KUKA KRL program: MyProgram_220().src

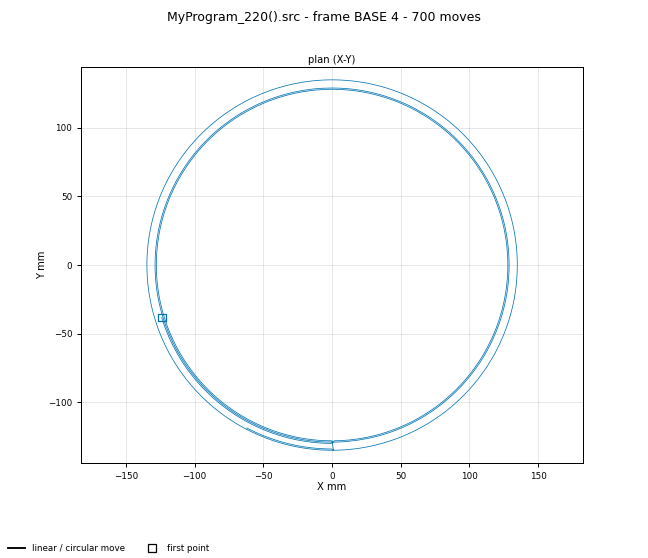
[picture p0: tool path of MyProgram_220().src in frame BASE 4, 700 of 700 moves have a stored position in this frame; points joined in program order, loops and branches not executed]
&ACCESS RVP
&REL 1
&PARAM TEMPLATE = C:\KRC\Roboter\Template\vorgabe
&PARAM EDITMASK = *
DEF MyProgram_220()
; ---- Setting reference (Base) ----
$BASE = BASE_DATA[4]

; --------------------------
; ---- Setting tool (TCP) ----
$TOOL = TOOL_DATA[3]
; --------------------------

$VEL.CP = VEL_APROX_PRINT
Startdeposition()
$VEL.CP = VEL_PRINT
LIN {X -124.0499,Y -38.1824,Z 153,A -164.431,B 20.1252,C -0.668,E1 19.9831,E2 612.3384} C_DIS
LIN {X -122.2235,Y -43.678,Z 153,A -161.8413,B 20.1254,C -0.6617,E1 19.9854,E2 609.7482} C_DIS
LIN {X -120.9472,Y -47.0955,Z 153,A -160.3023,B 20.1256,C -0.6544,E1 19.987,E2 608.2196} C_DIS
LIN {X -119.759,Y -50.0398,Z 153,A -158.8735,B 20.1257,C -0.6515,E1 19.9885,E2 606.7893} C_DIS
LIN {X -118.4765,Y -53.0047,Z 153,A -157.3393,B 20.1257,C -0.6515,E1 19.9902,E2 605.2441} C_DIS
LIN {X -116.9818,Y -56.2275,Z 153,A -155.8456,B 20.1259,C -0.6444,E1 19.992,E2 603.761} C_DIS
LIN {X -115.591,Y -59.0333,Z 153,A -154.3618,B 20.1259,C -0.6444,E1 19.9939,E2 602.2669} C_DIS
LIN {X -112.2722,Y -65.1279,Z 153,A -151.3304,B 20.1262,C -0.635,E1 19.998,E2 599.2428} C_DIS
LIN {X -110.2468,Y -68.5007,Z 153,A -149.5687,B 20.1263,C -0.6315,E1 20.0005,E2 597.48} C_DIS
LIN {X -107.8897,Y -72.1562,Z 153,A -147.8172,B 20.1267,C -0.6202,E1 20.0032,E2 595.7503} C_DIS
LIN {X -106.0602,Y -74.8192,Z 153,A -146.138,B 20.1265,C -0.6263,E1 20.0059,E2 594.0426} C_DIS
LIN {X -103.646,Y -78.1293,Z 153,A -144.4345,B 20.1267,C -0.6179,E1 20.0087,E2 592.3532} C_DIS
LIN {X -101.177,Y -81.3013,Z 153,A -142.5934,B 20.1267,C -0.6163,E1 20.0119,E2 590.5058} C_DIS
LIN {X -99.0599,Y -83.8683,Z 153,A -141.0774,B 20.1268,C -0.6147,E1 20.0146,E2 588.9855} C_DIS
LIN {X -96.3177,Y -87.0039,Z 153,A -139.1751,B 20.1268,C -0.6131,E1 20.0182,E2 587.0772} C_DIS
LIN {X -93.3696,Y -90.16,Z 153,A -137.2715,B 20.127,C -0.6089,E1 20.0218,E2 585.1754} C_DIS
LIN {X -88.6302,Y -94.8219,Z 153,A -134.3468,B 20.1272,C -0.6024,E1 20.0277,E2 582.254} C_DIS
LIN {X -86.2647,Y -96.9806,Z 153,A -132.8941,B 20.1272,C -0.6012,E1 20.0307,E2 580.7976} C_DIS
LIN {X -82.9316,Y -99.8452,Z 153,A -130.925,B 20.1272,C -0.5986,E1 20.0349,E2 578.8263} C_DIS
LIN {X -79.669,Y -102.4674,Z 153,A -129.0942,B 20.1274,C -0.5947,E1 20.0389,E2 576.9986} C_DIS
LIN {X -76.0312,Y -105.1949,Z 153,A -126.47,B 20.1268,C -0.6155,E1 20.045,E2 574.3017} C_DIS
LIN {X -71.6372,Y -108.2354,Z 153,A -125.0313,B 20.1279,C -0.5755,E1 20.0481,E2 572.9738} C_DIS
LIN {X -65.749,Y -111.9096,Z 153,A -121.6773,B 20.1278,C -0.5823,E1 20.0562,E2 569.5867} C_DIS
LIN {X -61.9654,Y -114.0484,Z 153,A -119.6951,B 20.1278,C -0.5822,E1 20.061,E2 567.5976} C_DIS
LIN {X -58.1719,Y -116.0295,Z 153,A -117.7274,B 20.1278,C -0.5829,E1 20.0659,E2 565.621} C_DIS
LIN {X -53.9421,Y -118.0541,Z 153,A -115.5017,B 20.1276,C -0.5867,E1 20.0716,E2 563.377} C_DIS
LIN {X -50.8123,Y -119.4344,Z 153,A -113.9211,B 20.1276,C -0.588,E1 20.0757,E2 561.7882} C_DIS
LIN {X -47.3478,Y -120.8491,Z 153,A -112.8761,B 20.1283,C -0.5621,E1 20.0782,E2 560.8158} C_DIS
LIN {X -43.644,Y -122.2357,Z 153,A -110.9408,B 20.1281,C -0.568,E1 20.0834,E2 558.8581} C_DIS
LIN {X -40.3205,Y -123.3734,Z 153,A -109.2108,B 20.128,C -0.574,E1 20.088,E2 557.1068} C_DIS
LIN {X -36.084,Y -124.6769,Z 153,A -107.4194,B 20.1282,C -0.5659,E1 20.0927,E2 555.335} C_DIS
LIN {X -32.6503,Y -125.6214,Z 153,A -105.6991,B 20.1281,C -0.5709,E1 20.0974,E2 553.5969} C_DIS
LIN {X -28.2074,Y -126.6929,Z 153,A -103.5651,B 20.128,C -0.5746,E1 20.1033,E2 551.4486} C_DIS
LIN {X -23.1298,Y -127.7159,Z 153,A -100.8212,B 20.1275,C -0.5924,E1 20.111,E2 548.6491} C_DIS
LIN {X -17.8854,Y -128.5559,Z 153,A -98.8039,B 20.1279,C -0.5784,E1 20.1164,E2 546.6708} C_DIS
LIN {X -14.3127,Y -129.0024,Z 153,A -97.7565,B 20.1285,C -0.5559,E1 20.1192,E2 545.6878} C_DIS
LIN {X -9.5222,Y -129.4436,Z 153,A -95.2617,B 20.1281,C -0.5709,E1 20.1262,E2 543.1478} C_DIS
LIN {X -4.67,Y -129.7099,Z 153,A -93.267,B 20.1282,C -0.5648,E1 20.1317,E2 541.1703} C_DIS
LIN {X -0.7047,Y -129.7915,Z 153,A -91.6167,B 20.1283,C -0.561,E1 20.1363,E2 539.5311} C_DIS
LIN {X -0.7047,Y -129.7915,Z 153,A -91.6167,B 20.1283,C -0.561,E1 20.1363,E2 539.5311} C_DIS
Enddeposition()
LIN {X 0.8922,Y -128.8473,Z 153,A -90.561,B 18.6911,C -0.3834,E1 18.6972,E2 538.8726} C_DIS
Startdeposition()
$VEL.CP = VEL_PRINT
LIN {X -1.7978,Y -128.8411,Z 153,A -92.3931,B 18.6916,C -0.3592,E1 18.6919,E2 540.7802} C_DIS
LIN {X -4.9626,Y -128.7576,Z 153,A -94.0816,B 18.6918,C -0.3487,E1 18.6871,E2 542.502} C_DIS
LIN {X -8.6262,Y -128.566,Z 153,A -95.4711,B 18.6916,C -0.3576,E1 18.6833,E2 543.8641} C_DIS
LIN {X -11.8778,Y -128.3052,Z 153,A -97.4568,B 18.692,C -0.3381,E1 18.6776,E2 545.9123} C_DIS
LIN {X -16.8123,Y -127.7516,Z 153,A -99.0184,B 18.6915,C -0.3623,E1 18.6735,E2 547.3997} C_DIS
LIN {X -20.6153,Y -127.1946,Z 153,A -100.8214,B 18.6915,C -0.3593,E1 18.6684,E2 549.2142} C_DIS
LIN {X -23.6637,Y -126.6626,Z 153,A -102.3077,B 18.6916,C -0.3558,E1 18.6643,E2 550.7136} C_DIS
LIN {X -28.0145,Y -125.7726,Z 153,A -104.178,B 18.6916,C -0.3606,E1 18.6593,E2 552.5722} C_DIS
LIN {X -31.1189,Y -125.0401,Z 153,A -105.392,B 18.6914,C -0.3688,E1 18.656,E2 553.7625} C_DIS
LIN {X -34.3257,Y -124.1972,Z 153,A -106.9978,B 18.6914,C -0.365,E1 18.6516,E2 555.3838} C_DIS
LIN {X -37.1865,Y -123.3714,Z 153,A -108.3483,B 18.6914,C -0.365,E1 18.648,E2 556.7375} C_DIS
LIN {X -40.6641,Y -122.2681,Z 153,A -109.8927,B 18.6914,C -0.3691,E1 18.6439,E2 558.2728} C_DIS
LIN {X -43.8363,Y -121.167,Z 153,A -111.4208,B 18.6914,C -0.3691,E1 18.6399,E2 559.8049} C_DIS
LIN {X -50.8161,Y -118.4097,Z 153,A -114.8178,B 18.6914,C -0.3702,E1 18.6311,E2 563.2088} C_DIS
LIN {X -54.652,Y -116.69,Z 153,A -116.9427,B 18.6915,C -0.3631,E1 18.6256,E2 565.363} C_DIS
LIN {X -59.4438,Y -114.3228,Z 153,A -119.0566,B 18.6913,C -0.3755,E1 18.6204,E2 567.4459} C_DIS
LIN {X -63.0684,Y -112.365,Z 153,A -120.8296,B 18.6912,C -0.38,E1 18.6161,E2 569.2117} C_DIS
LIN {X -67.2669,Y -109.9031,Z 153,A -123.1372,B 18.6912,C -0.378,E1 18.6105,E2 571.5353} C_DIS
LIN {X -71.1021,Y -107.462,Z 153,A -125.0591,B 18.6911,C -0.3847,E1 18.6061,E2 573.445} C_DIS
LIN {X -74.9299,Y -104.8285,Z 153,A -127.1982,B 18.6911,C -0.3854,E1 18.6012,E2 575.5916} C_DIS
LIN {X -78.3456,Y -102.3009,Z 153,A -128.9712,B 18.6909,C -0.3928,E1 18.5972,E2 577.3502} C_DIS
LIN {X -81.75,Y -99.6018,Z 153,A -131.0814,B 18.6909,C -0.39,E1 18.5926,E2 579.4801} C_DIS
LIN {X -85.1235,Y -96.7346,Z 153,A -132.9003,B 18.6909,C -0.399,E1 18.5888,E2 581.2806} C_DIS
LIN {X -91.5255,Y -90.7005,Z 153,A -136.9673,B 18.6908,C -0.4014,E1 18.5806,E2 585.3631} C_DIS
LIN {X -94.7022,Y -87.3787,Z 153,A -139.0611,B 18.6908,C -0.4041,E1 18.5765,E2 587.4613} C_DIS
LIN {X -97.6736,Y -84.0439,Z 153,A -141.0409,B 18.6906,C -0.4087,E1 18.5729,E2 589.4388} C_DIS
LIN {X -101.5319,Y -79.3402,Z 153,A -143.629,B 18.6904,C -0.419,E1 18.5684,E2 592.0113} C_DIS
LIN {X -103.7936,Y -76.357,Z 153,A -145.4466,B 18.6904,C -0.4177,E1 18.5653,E2 593.845} C_DIS
LIN {X -106.3954,Y -72.6884,Z 153,A -147.4209,B 18.6903,C -0.4234,E1 18.5621,E2 595.8146} C_DIS
LIN {X -108.6997,Y -69.1953,Z 153,A -149.3063,B 18.6903,C -0.4273,E1 18.5593,E2 597.7011} C_DIS
LIN {X -110.9258,Y -65.5675,Z 153,A -151.256,B 18.6901,C -0.4302,E1 18.5565,E2 599.6554} C_DIS
LIN {X -112.4474,Y -62.9218,Z 153,A -152.7042,B 18.6901,C -0.4306,E1 18.5545,E2 601.1128} C_DIS
LIN {X -114.4576,Y -59.1871,Z 153,A -154.5413,B 18.69,C -0.4373,E1 18.5521,E2 602.9423} C_DIS
LIN {X -116.1156,Y -55.8596,Z 153,A -155.9219,B 18.6897,C -0.4511,E1 18.5504,E2 604.2898} C_DIS
LIN {X -117.4691,Y -52.9543,Z 153,A -157.4356,B 18.6897,C -0.452,E1 18.5486,E2 605.8121} C_DIS
LIN {X -118.5866,Y -50.407,Z 153,A -158.9047,B 18.6897,C -0.4475,E1 18.547,E2 607.3065} C_DIS
LIN {X -119.9416,Y -47.0875,Z 153,A -160.199,B 18.6894,C -0.4622,E1 18.5457,E2 608.5646} C_DIS
LIN {X -121.0477,Y -44.1669,Z 153,A -161.8114,B 18.6894,C -0.4586,E1 18.5441,E2 610.2009} C_DIS
LIN {X -122.7867,Y -39.0704,Z 153,A -164.1851,B 18.6894,C -0.4662,E1 18.542,E2 612.5694} C_DIS
LIN {X -123.9311,Y -35.2775,Z 153,A -165.9601,B 18.6892,C -0.4709,E1 18.5406,E2 614.3438} C_DIS
LIN {X -124.8345,Y -31.9292,Z 153,A -167.5525,B 18.6892,C -0.4738,E1 18.5395,E2 615.9399} C_DIS
LIN {X -125.8011,Y -27.8864,Z 153,A -169.46,B 18.689,C -0.4773,E1 18.5383,E2 617.8519} C_DIS
LIN {X -126.5739,Y -24.1273,Z 153,A -171.1769,B 18.689,C -0.4821,E1 18.5373,E2 619.5676} C_DIS
LIN {X -127.2655,Y -20.1692,Z 153,A -172.7668,B 18.6886,C -0.4941,E1 18.5366,E2 621.1327} C_DIS
LIN {X -127.7311,Y -16.968,Z 153,A -174.4022,B 18.6886,C -0.4919,E1 18.536,E2 622.7886} C_DIS
LIN {X -128.1554,Y -13.3956,Z 153,A -176.0902,B 18.6886,C -0.4938,E1 18.5354,E2 624.4845} C_DIS
LIN {X -128.5161,Y -9.3142,Z 153,A -177.7957,B 18.6884,C -0.5034,E1 18.5351,E2 626.1742} C_DIS
LIN {X -128.7367,Y -5.4997,Z 153,A -179.3666,B 18.6881,C -0.5129,E1 18.5348,E2 627.7281} C_DIS
LIN {X -128.8292,Y -2.5182,Z 153,A 179.1207,B 18.6881,C -0.5108,E1 18.5348,E2 629.2602} C_DIS
LIN {X -128.8489,Y 1.1038,Z 153,A 177.6722,B 18.6879,C -0.5212,E1 18.5348,E2 630.6879} C_DIS
LIN {X -128.792,Y 3.9938,Z 153,A 176.1149,B 18.688,C -0.5161,E1 18.5348,E2 632.2743} C_DIS
LIN {X -128.5815,Y 8.3752,Z 153,A 173.9578,B 18.688,C -0.5152,E1 18.5352,E2 634.4519} C_DIS
LIN {X -128.3292,Y 11.6281,Z 153,A 172.6535,B 18.6878,C -0.5246,E1 18.5355,E2 635.7376} C_DIS
LIN {X -127.8595,Y 15.9868,Z 153,A 170.6979,B 18.6877,C -0.5304,E1 18.5361,E2 637.691} C_DIS
LIN {X -127.3978,Y 19.3149,Z 153,A 169.2335,B 18.6875,C -0.536,E1 18.5367,E2 639.1497} C_DIS
LIN {X -126.6839,Y 23.5521,Z 153,A 167.3093,B 18.6874,C -0.5415,E1 18.5377,E2 641.0727} C_DIS
LIN {X -125.9625,Y 27.1388,Z 153,A 165.7576,B 18.6871,C -0.549,E1 18.5385,E2 642.6134} C_DIS
LIN {X -125.0826,Y 30.9515,Z 153,A 163.8735,B 18.6871,C -0.5494,E1 18.5398,E2 644.5113} C_DIS
LIN {X -123.9507,Y 35.2073,Z 153,A 161.3522,B 18.6875,C -0.5367,E1 18.5417,E2 647.0929} C_DIS
LIN {X -122.4844,Y 40.0115,Z 153,A 159.7319,B 18.6867,C -0.5638,E1 18.543,E2 648.6408} C_DIS
LIN {X -121.2971,Y 43.4752,Z 153,A 158.0558,B 18.6867,C -0.567,E1 18.5446,E2 650.3199} C_DIS
LIN {X -119.855,Y 47.3102,Z 153,A 156.2801,B 18.6864,C -0.5739,E1 18.5464,E2 652.0876} C_DIS
LIN {X -118.5641,Y 50.4591,Z 153,A 154.6433,B 18.6864,C -0.5742,E1 18.5481,E2 653.7362} C_DIS
LIN {X -117.0382,Y 53.8991,Z 153,A 152.5033,B 18.6867,C -0.5634,E1 18.5507,E2 655.9261} C_DIS
LIN {X -115.0458,Y 58.0318,Z 153,A 151.1702,B 18.6858,C -0.5929,E1 18.5522,E2 657.1765} C_DIS
LIN {X -113.5082,Y 60.9869,Z 153,A 149.4584,B 18.686,C -0.5893,E1 18.5545,E2 658.9123} C_DIS
LIN {X -111.3388,Y 64.8638,Z 153,A 147.5706,B 18.6857,C -0.5977,E1 18.5571,E2 660.7873} C_DIS
LIN {X -107.9641,Y 70.337,Z 153,A 144.6774,B 18.6855,C -0.6042,E1 18.5614,E2 663.6801} C_DIS
LIN {X -105.8908,Y 73.4213,Z 153,A 142.8887,B 18.6855,C -0.604,E1 18.5642,E2 665.4818} C_DIS
LIN {X -103.5804,Y 76.647,Z 153,A 141.0878,B 18.6854,C -0.6073,E1 18.5672,E2 667.2843} C_DIS
LIN {X -100.8812,Y 80.1655,Z 153,A 139.1659,B 18.6852,C -0.614,E1 18.5704,E2 669.1977} C_DIS
LIN {X -98.2339,Y 83.3883,Z 153,A 137.2838,B 18.6851,C -0.6177,E1 18.5738,E2 671.0803} C_DIS
LIN {X -95.3863,Y 86.6312,Z 153,A 135.3556,B 18.6849,C -0.622,E1 18.5774,E2 673.0069} C_DIS
LIN {X -92.3221,Y 89.8903,Z 153,A 133.3182,B 18.6849,C -0.625,E1 18.5813,E2 675.047} C_DIS
LIN {X -89.3268,Y 92.8677,Z 153,A 131.4363,B 18.6847,C -0.6291,E1 18.5851,E2 676.9269} C_DIS
LIN {X -86.4368,Y 95.5627,Z 153,A 129.7432,B 18.6845,C -0.6352,E1 18.5885,E2 678.6103} C_DIS
LIN {X -83.4105,Y 98.2151,Z 153,A 127.9104,B 18.6845,C -0.6375,E1 18.5924,E2 680.4457} C_DIS
LIN {X -80.1785,Y 100.8708,Z 153,A 126.018,B 18.6843,C -0.6402,E1 18.5965,E2 682.3394} C_DIS
LIN {X -76.6483,Y 103.5794,Z 153,A 123.9948,B 18.6843,C -0.6426,E1 18.6011,E2 684.3652} C_DIS
LIN {X -74.3543,Y 105.2376,Z 153,A 122.5318,B 18.6844,C -0.6379,E1 18.6044,E2 685.8496} C_DIS
LIN {X -71.6808,Y 107.0766,Z 153,A 120.9403,B 18.6844,C -0.6355,E1 18.6082,E2 687.4562} C_DIS
LIN {X -68.3675,Y 109.222,Z 153,A 119.4648,B 18.6841,C -0.6482,E1 18.6116,E2 688.8982} C_DIS
LIN {X -64.3417,Y 111.641,Z 153,A 117.4252,B 18.6839,C -0.6534,E1 18.6165,E2 690.9298} C_DIS
LIN {X -60.6816,Y 113.6722,Z 153,A 115.6579,B 18.6837,C -0.6597,E1 18.6208,E2 692.6845} C_DIS
LIN {X -57.2859,Y 115.4185,Z 153,A 113.919,B 18.6837,C -0.6609,E1 18.6251,E2 694.426} C_DIS
LIN {X -53.7581,Y 117.1034,Z 153,A 112.164,B 18.6836,C -0.6628,E1 18.6295,E2 696.1811} C_DIS
LIN {X -50.4862,Y 118.5524,Z 153,A 110.6594,B 18.6834,C -0.668,E1 18.6334,E2 697.6743} C_DIS
LIN {X -47.2881,Y 119.8636,Z 153,A 108.9988,B 18.6834,C -0.6656,E1 18.6377,E2 699.3474} C_DIS
LIN {X -43.8521,Y 121.1613,Z 153,A 107.4552,B 18.6834,C -0.6707,E1 18.6417,E2 700.8793} C_DIS
LIN {X -40.8666,Y 122.2006,Z 153,A 106.1838,B 18.6831,C -0.6771,E1 18.645,E2 702.1342} C_DIS
LIN {X -38.5993,Y 122.9372,Z 153,A 104.8373,B 18.6834,C -0.668,E1 18.6487,E2 703.5122} C_DIS
LIN {X -35.0688,Y 123.9894,Z 153,A 103.459,B 18.683,C -0.6789,E1 18.6523,E2 704.8597} C_DIS
LIN {X -32.3809,Y 124.7198,Z 153,A 101.839,B 18.6835,C -0.6664,E1 18.6568,E2 706.5219} C_DIS
LIN {X -27.7778,Y 125.8246,Z 153,A 99.5881,B 18.6835,C -0.663,E1 18.663,E2 708.7876} C_DIS
LIN {X -24.3768,Y 126.5262,Z 153,A 98.4114,B 18.6831,C -0.6772,E1 18.6661,E2 709.9215} C_DIS
LIN {X -20.9195,Y 127.1438,Z 153,A 96.8722,B 18.6831,C -0.6791,E1 18.6703,E2 711.4571} C_DIS
LIN {X -14.7385,Y 128.0085,Z 153,A 94.1208,B 18.6829,C -0.6814,E1 18.6779,E2 714.204} C_DIS
LIN {X -11.298,Y 128.3575,Z 153,A 92.0352,B 18.6836,C -0.6623,E1 18.6839,E2 716.3507} C_DIS
LIN {X -7.0803,Y 128.6599,Z 153,A 90.7429,B 18.6828,C -0.6841,E1 18.6873,E2 717.5754} C_DIS
LIN {X 0.1516,Y 128.8544,Z 153,A 86.6454,B 18.6839,C -0.6528,E1 18.699,E2 721.7707} C_DIS
LIN {X 5.794,Y 128.7246,Z 153,A 84.9882,B 18.6829,C -0.6838,E1 18.7034,E2 723.3306} C_DIS
LIN {X 11.8096,Y 128.3118,Z 153,A 82.0309,B 18.6832,C -0.6734,E1 18.7117,E2 726.3183} C_DIS
LIN {X 16.2936,Y 127.8195,Z 153,A 80.2191,B 18.683,C -0.6801,E1 18.7166,E2 728.1075} C_DIS
LIN {X 19.5858,Y 127.3559,Z 153,A 78.8596,B 18.6828,C -0.684,E1 18.7203,E2 729.4529} C_DIS
LIN {X 23.1661,Y 126.7543,Z 153,A 77.167,B 18.683,C -0.6805,E1 18.725,E2 731.1541} C_DIS
LIN {X 27.1118,Y 125.9684,Z 153,A 75.6191,B 18.6827,C -0.6886,E1 18.7292,E2 732.6741} C_DIS
LIN {X 30.0875,Y 125.2909,Z 153,A 73.9169,B 18.6832,C -0.6749,E1 18.7339,E2 734.4156} C_DIS
LIN {X 33.9159,Y 124.3114,Z 153,A 72.277,B 18.6831,C -0.6781,E1 18.7383,E2 736.0419} C_DIS
LIN {X 36.8949,Y 123.4598,Z 153,A 70.7652,B 18.6833,C -0.6721,E1 18.7424,E2 737.569} C_DIS
LIN {X 40.5844,Y 122.2946,Z 153,A 69.2515,B 18.683,C -0.6784,E1 18.7464,E2 739.0589} C_DIS
LIN {X 43.0947,Y 121.4343,Z 153,A 66.983,B 18.6845,C -0.6366,E1 18.7527,E2 741.4511} C_DIS
LIN {X 49.3151,Y 119.0427,Z 153,A 65.0437,B 18.6833,C -0.6719,E1 18.7574,E2 743.2745} C_DIS
LIN {X 53.1423,Y 117.385,Z 153,A 63.1989,B 18.6833,C -0.6702,E1 18.7621,E2 745.1185} C_DIS
LIN {X 56.4826,Y 115.8148,Z 153,A 61.4722,B 18.6835,C -0.6649,E1 18.7665,E2 746.8553} C_DIS
LIN {X 60.0312,Y 114.0144,Z 153,A 59.931,B 18.6833,C -0.6713,E1 18.7702,E2 748.3707} C_DIS
LIN {X 66.8158,Y 110.178,Z 153,A 56.2335,B 18.6838,C -0.6575,E1 18.7793,E2 752.096} C_DIS
LIN {X 71.3155,Y 107.3204,Z 153,A 53.8497,B 18.6839,C -0.6532,E1 18.7848,E2 754.4823} C_DIS
LIN {X 74.8349,Y 104.8964,Z 153,A 51.9744,B 18.6839,C -0.651,E1 18.7891,E2 756.3555} C_DIS
LIN {X 78.4833,Y 102.1956,Z 153,A 49.9711,B 18.6841,C -0.6481,E1 18.7936,E2 758.358} C_DIS
LIN {X 81.766,Y 99.5887,Z 153,A 48.15,B 18.6841,C -0.6463,E1 18.7975,E2 760.1752} C_DIS
LIN {X 85.0534,Y 96.7966,Z 153,A 46.2322,B 18.6843,C -0.6426,E1 18.8016,E2 762.094} C_DIS
LIN {X 88.3958,Y 93.7533,Z 153,A 44.1218,B 18.6845,C -0.6347,E1 18.8059,E2 764.2172} C_DIS
LIN {X 91.755,Y 90.469,Z 153,A 42.1091,B 18.6845,C -0.6333,E1 18.8099,E2 766.2225} C_DIS
LIN {X 94.6799,Y 87.403,Z 153,A 40.2376,B 18.6847,C -0.6297,E1 18.8135,E2 768.0939} C_DIS
LIN {X 97.4633,Y 84.2881,Z 153,A 38.3922,B 18.6848,C -0.626,E1 18.8169,E2 769.9393} C_DIS
LIN {X 100.483,Y 80.6645,Z 153,A 36.3264,B 18.6849,C -0.6224,E1 18.8205,E2 772.0032} C_DIS
LIN {X 103.11,Y 77.2786,Z 153,A 34.5596,B 18.6849,C -0.6233,E1 18.8235,E2 773.7555} C_DIS
LIN {X 107.3136,Y 71.3258,Z 153,A 31.2168,B 18.6853,C -0.6112,E1 18.8289,E2 777.1132} C_DIS
LIN {X 109.1635,Y 68.4615,Z 153,A 29.4966,B 18.6856,C -0.5993,E1 18.8315,E2 778.8584} C_DIS
LIN {X 110.8629,Y 65.6738,Z 153,A 28.3684,B 18.6854,C -0.6083,E1 18.833,E2 779.9506} C_DIS
LIN {X 112.8659,Y 62.1682,Z 153,A 26.4796,B 18.6856,C -0.5999,E1 18.8356,E2 781.8521} C_DIS
LIN {X 114.5817,Y 58.9434,Z 153,A 25.0921,B 18.6855,C -0.605,E1 18.8374,E2 783.2138} C_DIS
LIN {X 117.1547,Y 53.6472,Z 153,A 22.2619,B 18.686,C -0.5893,E1 18.8409,E2 786.0715} C_DIS
LIN {X 118.447,Y 50.7298,Z 153,A 20.6234,B 18.6863,C -0.5766,E1 18.8427,E2 787.737} C_DIS
LIN {X 119.7997,Y 47.4516,Z 153,A 19.3063,B 18.6862,C -0.5825,E1 18.844,E2 789.026} C_DIS
LIN {X 120.9848,Y 44.3414,Z 153,A 17.7597,B 18.6864,C -0.5756,E1 18.8455,E2 790.582} C_DIS
LIN {X 122.342,Y 40.4419,Z 153,A 16.1053,B 18.6864,C -0.5776,E1 18.847,E2 792.2176} C_DIS
LIN {X 123.5409,Y 36.6179,Z 153,A 14.3858,B 18.6864,C -0.5748,E1 18.8484,E2 793.9319} C_DIS
LIN {X 124.3314,Y 33.8407,Z 153,A 12.9628,B 18.6867,C -0.5655,E1 18.8495,E2 795.3728} C_DIS
LIN {X 125.261,Y 30.2117,Z 153,A 10.9903,B 18.6872,C -0.5482,E1 18.8508,E2 797.383} C_DIS
LIN {X 126.135,Y 26.3337,Z 153,A 9.6959,B 18.6868,C -0.5619,E1 18.8515,E2 798.6248} C_DIS
LIN {X 126.7331,Y 23.2846,Z 153,A 8.2849,B 18.6869,C -0.5565,E1 18.8523,E2 800.041} C_DIS
LIN {X 127.2322,Y 20.3842,Z 153,A 6.5211,B 18.6876,C -0.5343,E1 18.8531,E2 801.8594} C_DIS
LIN {X 127.8062,Y 16.3951,Z 153,A 5.2549,B 18.6871,C -0.5499,E1 18.8535,E2 803.0669} C_DIS
LIN {X 128.5105,Y 9.3908,Z 153,A 2.4485,B 18.6871,C -0.5533,E1 18.8543,E2 805.8399} C_DIS
LIN {X 128.8357,Y 2.1236,Z 153,A -0.7464,B 18.6873,C -0.5448,E1 18.8547,E2 809.035} C_DIS
LIN {X 128.7821,Y -4.335,Z 153,A -4.0261,B 18.688,C -0.5193,E1 18.8546,E2 812.3668} C_DIS
LIN {X 128.3422,Y -11.4815,Z 153,A -7.2602,B 18.6883,C -0.5074,E1 18.8539,E2 815.6115} C_DIS
LIN {X 127.8619,Y -15.9669,Z 153,A -9.1185,B 18.6883,C -0.5071,E1 18.8533,E2 817.4555} C_DIS
LIN {X 127.4527,Y -18.9583,Z 153,A -10.6936,B 18.6886,C -0.4935,E1 18.8527,E2 819.0598} C_DIS
LIN {X 126.6103,Y -23.9373,Z 153,A -12.5459,B 18.6884,C -0.5025,E1 18.8518,E2 820.8695} C_DIS
LIN {X 125.8028,Y -27.8786,Z 153,A -14.5783,B 18.6888,C -0.4871,E1 18.8506,E2 822.9332} C_DIS
LIN {X 125.0008,Y -31.2738,Z 153,A -15.8685,B 18.6886,C -0.493,E1 18.8498,E2 824.1952} C_DIS
LIN {X 124.0369,Y -34.899,Z 153,A -17.399,B 18.6886,C -0.4934,E1 18.8487,E2 825.712} C_DIS
LIN {X 122.9845,Y -38.4507,Z 153,A -19.4112,B 18.6891,C -0.4737,E1 18.847,E2 827.7696} C_DIS
LIN {X 121.5142,Y -42.8698,Z 153,A -21.2595,B 18.6891,C -0.4765,E1 18.8454,E2 829.595} C_DIS
LIN {X 119.7651,Y -47.5376,Z 153,A -23.4411,B 18.6891,C -0.4713,E1 18.8432,E2 831.7759} C_DIS
LIN {X 118.3665,Y -50.916,Z 153,A -24.8633,B 18.6891,C -0.4748,E1 18.8417,E2 833.1766} C_DIS
LIN {X 117.1454,Y -53.6672,Z 153,A -26.5105,B 18.6895,C -0.4584,E1 18.8398,E2 834.8622} C_DIS
LIN {X 115.2522,Y -57.623,Z 153,A -28.7299,B 18.6899,C -0.442,E1 18.837,E2 837.116} C_DIS
LIN {X 113.6154,Y -60.7873,Z 153,A -30.032,B 18.6897,C -0.4488,E1 18.8353,E2 838.3875} C_DIS
LIN {X 111.463,Y -64.6492,Z 153,A -31.9535,B 18.6898,C -0.4451,E1 18.8327,E2 840.3067} C_DIS
LIN {X 109.2277,Y -68.3587,Z 153,A -33.9322,B 18.69,C -0.4377,E1 18.8298,E2 842.2945} C_DIS
LIN {X 106.9157,Y -71.9213,Z 153,A -35.806,B 18.69,C -0.4332,E1 18.8269,E2 844.1694} C_DIS
LIN {X 104.784,Y -74.9922,Z 153,A -37.4446,B 18.6901,C -0.4298,E1 18.8242,E2 845.8077} C_DIS
LIN {X 102.5622,Y -78.004,Z 153,A -39.1097,B 18.6902,C -0.4255,E1 18.8214,E2 847.4753} C_DIS
LIN {X 99.6794,Y -81.655,Z 153,A -41.0674,B 18.6902,C -0.4246,E1 18.818,E2 849.423} C_DIS
LIN {X 97.3996,Y -84.3615,Z 153,A -42.7538,B 18.6904,C -0.4162,E1 18.8149,E2 851.1248} C_DIS
LIN {X 94.1796,Y -87.9416,Z 153,A -44.7963,B 18.6904,C -0.415,E1 18.8111,E2 853.1587} C_DIS
LIN {X 91.1521,Y -91.0765,Z 153,A -46.6426,B 18.6904,C -0.4141,E1 18.8075,E2 854.997} C_DIS
LIN {X 88.6923,Y -93.4731,Z 153,A -48.2764,B 18.6907,C -0.4064,E1 18.8042,E2 856.6454} C_DIS
LIN {X 85.4273,Y -96.466,Z 153,A -50.1588,B 18.6907,C -0.4055,E1 18.8003,E2 858.5202} C_DIS
LIN {X 82.6432,Y -98.8618,Z 153,A -51.8268,B 18.6907,C -0.4006,E1 18.7967,E2 860.1944} C_DIS
LIN {X 79.8799,Y -101.108,Z 153,A -53.5052,B 18.6909,C -0.3936,E1 18.7931,E2 861.886} C_DIS
LIN {X 75.9801,Y -104.0705,Z 153,A -55.5271,B 18.6909,C -0.3953,E1 18.7886,E2 863.8924} C_DIS
LIN {X 72.5224,Y -106.5088,Z 153,A -57.4849,B 18.691,C -0.3887,E1 18.784,E2 865.8615} C_DIS
LIN {X 68.6992,Y -109.0135,Z 153,A -59.4393,B 18.691,C -0.3881,E1 18.7795,E2 867.8091} C_DIS
LIN {X 65.0563,Y -111.2261,Z 153,A -61.3563,B 18.6911,C -0.3839,E1 18.7749,E2 869.7309} C_DIS
LIN {X 61.4641,Y -113.2508,Z 153,A -63.5586,B 18.6914,C -0.3665,E1 18.7694,E2 871.9784} C_DIS
LIN {X 57.8986,Y -115.1136,Z 153,A -64.8895,B 18.6912,C -0.3815,E1 18.7662,E2 873.2577} C_DIS
LIN {X 54.8571,Y -116.5945,Z 153,A -66.4013,B 18.6912,C -0.3789,E1 18.7624,E2 874.7721} C_DIS
LIN {X 51.9098,Y -117.9363,Z 153,A -67.768,B 18.6912,C -0.3797,E1 18.7589,E2 876.1316} C_DIS
LIN {X 47.9256,Y -119.6087,Z 153,A -69.813,B 18.6913,C -0.3723,E1 18.7536,E2 878.1931} C_DIS
LIN {X 44.2185,Y -121.0291,Z 153,A -71.4368,B 18.6913,C -0.3756,E1 18.7494,E2 879.802} C_DIS
LIN {X 41.1968,Y -122.0906,Z 153,A -73.339,B 18.6917,C -0.3555,E1 18.7442,E2 881.7614} C_DIS
LIN {X 37.4971,Y -123.2764,Z 153,A -74.5826,B 18.6913,C -0.3722,E1 18.741,E2 882.95} C_DIS
LIN {X 34.0113,Y -124.2852,Z 153,A -76.3773,B 18.6915,C -0.3636,E1 18.7361,E2 884.7674} C_DIS
LIN {X 30.2742,Y -125.246,Z 153,A -78.3876,B 18.6917,C -0.3508,E1 18.7306,E2 886.8134} C_DIS
LIN {X 26.309,Y -126.14,Z 153,A -79.8338,B 18.6915,C -0.363,E1 18.7267,E2 888.219} C_DIS
LIN {X 17.449,Y -127.6681,Z 153,A -83.6764,B 18.6915,C -0.3661,E1 18.7162,E2 892.0464} C_DIS
LIN {X 9.4408,Y -128.5068,Z 153,A -87.3874,B 18.6915,C -0.3594,E1 18.7059,E2 895.775} C_DIS
LIN {X 4.7553,Y -128.7657,Z 153,A -89.4989,B 18.6916,C -0.3578,E1 18.6999,E2 897.8906} C_DIS
LIN {X 0.8922,Y -128.8473,Z 153,A -90.5575,B 18.6911,C -0.3823,E1 18.6972,E2 898.8726} C_DIS
Enddeposition()
LIN {X 0.8922,Y -128.8473,Z 153,A -90.5575,B 18.6911,C -0.3823,E1 18.6972,E2 898.8726} C_DIS
Startdeposition()
$VEL.CP = VEL_PRINT
LIN {X 1.5624,Y -127.9047,Z 153,A -89.64,B 17.5227,C -0.2683,E1 17.5287,E2 898.2231} C_DIS
LIN {X 6.2751,Y -127.7591,Z 153,A -87.8027,B 17.5227,C -0.2592,E1 17.5337,E2 896.4169} C_DIS
LIN {X 9.4059,Y -127.5667,Z 153,A -86.3309,B 17.5227,C -0.2621,E1 17.5379,E2 894.9364} C_DIS
LIN {X 12.2166,Y -127.3282,Z 153,A -85.0464,B 17.5227,C -0.2634,E1 17.5414,E2 893.6487} C_DIS
LIN {X 15.3093,Y -126.9935,Z 153,A -83.673,B 17.5227,C -0.2634,E1 17.5452,E2 892.2767} C_DIS
LIN {X 18.1453,Y -126.6193,Z 153,A -82.3008,B 17.5227,C -0.2674,E1 17.5491,E2 890.893} C_DIS
LIN {X 21.4662,Y -126.0994,Z 153,A -80.8299,B 17.5227,C -0.2672,E1 17.5531,E2 889.4251} C_DIS
LIN {X 24.507,Y -125.5441,Z 153,A -79.4012,B 17.5227,C -0.2698,E1 17.5571,E2 887.9903} C_DIS
LIN {X 27.6498,Y -124.8904,Z 153,A -78.0615,B 17.5227,C -0.2674,E1 17.5607,E2 886.661} C_DIS
LIN {X 30.7266,Y -124.1697,Z 153,A -76.6506,B 17.5227,C -0.2685,E1 17.5645,E2 885.2495} C_DIS
LIN {X 33.7547,Y -123.3807,Z 153,A -75.2428,B 17.5227,C -0.2701,E1 17.5683,E2 883.8398} C_DIS
LIN {X 37.1173,Y -122.4094,Z 153,A -73.6815,B 17.5227,C -0.2715,E1 17.5725,E2 882.2779} C_DIS
LIN {X 39.7454,Y -121.583,Z 153,A -72.3376,B 17.5225,C -0.2769,E1 17.5761,E2 880.92} C_DIS
LIN {X 42.7469,Y -120.5603,Z 153,A -71.0375,B 17.5225,C -0.2742,E1 17.5795,E2 879.6327} C_DIS
LIN {X 45.6876,Y -119.477,Z 153,A -69.6412,B 17.5225,C -0.2756,E1 17.5832,E2 878.236} C_DIS
LIN {X 48.6016,Y -118.3218,Z 153,A -68.1197,B 17.5225,C -0.2818,E1 17.5871,E2 876.6993} C_DIS
LIN {X 51.8383,Y -116.9383,Z 153,A -66.8123,B 17.5225,C -0.2741,E1 17.5904,E2 875.4219} C_DIS
LIN {X 54.6839,Y -115.6353,Z 153,A -65.2797,B 17.5225,C -0.2809,E1 17.5943,E2 873.8726} C_DIS
LIN {X 57.495,Y -114.2641,Z 153,A -63.888,B 17.5225,C -0.2827,E1 17.5978,E2 872.4806} C_DIS
LIN {X 59.9433,Y -112.9986,Z 153,A -62.616,B 17.5224,C -0.286,E1 17.601,E2 871.2028} C_DIS
LIN {X 62.9591,Y -111.3479,Z 153,A -61.1533,B 17.5224,C -0.2857,E1 17.6045,E2 869.7475} C_DIS
LIN {X 65.7569,Y -109.7188,Z 153,A -59.6681,B 17.5224,C -0.2895,E1 17.6081,E2 868.2565} C_DIS
LIN {X 68.4368,Y -108.0673,Z 153,A -58.347,B 17.5224,C -0.2887,E1 17.6112,E2 866.9444} C_DIS
LIN {X 70.7618,Y -106.5597,Z 153,A -57.0438,B 17.5223,C -0.2933,E1 17.6143,E2 865.6324} C_DIS
LIN {X 73.3534,Y -104.7927,Z 153,A -55.6339,B 17.5223,C -0.2961,E1 17.6175,E2 864.2203} C_DIS
LIN {X 75.8966,Y -102.9652,Z 153,A -54.2421,B 17.5222,C -0.2984,E1 17.6207,E2 862.8281} C_DIS
LIN {X 78.7023,Y -100.8375,Z 153,A -52.5161,B 17.522,C -0.3071,E1 17.6245,E2 861.0826} C_DIS
LIN {X 82.2144,Y -97.9943,Z 153,A -50.6306,B 17.522,C -0.3062,E1 17.6286,E2 859.2108} C_DIS
LIN {X 85.1757,Y -95.4318,Z 153,A -48.8827,B 17.522,C -0.3097,E1 17.6322,E2 857.4615} C_DIS
LIN {X 88.056,Y -92.7813,Z 153,A -47.1347,B 17.522,C -0.3134,E1 17.6358,E2 855.7119} C_DIS
LIN {X 90.8736,Y -90.0228,Z 153,A -45.3648,B 17.5219,C -0.3176,E1 17.6393,E2 853.9391} C_DIS
LIN {X 93.7104,Y -87.0659,Z 153,A -43.5722,B 17.5219,C -0.3203,E1 17.6427,E2 852.1492} C_DIS
LIN {X 96.3308,Y -84.1575,Z 153,A -41.7492,B 17.5217,C -0.3272,E1 17.6461,E2 850.3156} C_DIS
LIN {X 98.9944,Y -81.0075,Z 153,A -39.9222,B 17.5217,C -0.3309,E1 17.6494,E2 848.4885} C_DIS
LIN {X 101.4282,Y -77.939,Z 153,A -38.1645,B 17.5215,C -0.3355,E1 17.6524,E2 846.728} C_DIS
LIN {X 103.6605,Y -74.9441,Z 153,A -36.6248,B 17.5215,C -0.3348,E1 17.6549,E2 845.2016} C_DIS
LIN {X 105.4763,Y -72.3661,Z 153,A -35.2254,B 17.5215,C -0.338,E1 17.6572,E2 843.8019} C_DIS
LIN {X 107.2194,Y -69.7575,Z 153,A -33.8339,B 17.5215,C -0.3412,E1 17.6593,E2 842.4099} C_DIS
LIN {X 108.7034,Y -67.4218,Z 153,A -32.5352,B 17.5213,C -0.3468,E1 17.6613,E2 841.1025} C_DIS
LIN {X 110.8638,Y -63.8076,Z 153,A -30.6192,B 17.5213,C -0.3531,E1 17.664,E2 839.1804} C_DIS
LIN {X 112.6371,Y -60.6217,Z 153,A -29.0731,B 17.5212,C -0.3543,E1 17.666,E2 837.6421} C_DIS
LIN {X 114.0975,Y -57.8222,Z 153,A -27.7059,B 17.5212,C -0.3565,E1 17.6678,E2 836.2783} C_DIS
LIN {X 115.4781,Y -55.0129,Z 153,A -26.2658,B 17.521,C -0.3619,E1 17.6695,E2 834.8318} C_DIS
LIN {X 116.9386,Y -51.8376,Z 153,A -24.8082,B 17.521,C -0.3623,E1 17.6712,E2 833.3846} C_DIS
LIN {X 118.1728,Y -48.9585,Z 153,A -23.3721,B 17.521,C -0.3676,E1 17.6728,E2 831.9426} C_DIS
LIN {X 119.3359,Y -46.0507,Z 153,A -21.9823,B 17.5208,C -0.3712,E1 17.6742,E2 830.5523} C_DIS
LIN {X 120.6724,Y -42.4276,Z 153,A -20.0786,B 17.5206,C -0.383,E1 17.676,E2 828.6257} C_DIS
LIN {X 121.9388,Y -38.6349,Z 153,A -18.5512,B 17.5206,C -0.3782,E1 17.6773,E2 827.1266} C_DIS
LIN {X 122.8538,Y -35.6188,Z 153,A -17.0953,B 17.5206,C -0.3841,E1 17.6784,E2 825.6634} C_DIS
LIN {X 123.6898,Y -32.598,Z 153,A -15.705,B 17.5205,C -0.3878,E1 17.6795,E2 824.2727} C_DIS
LIN {X 124.4515,Y -29.5577,Z 153,A -14.315,B 17.5205,C -0.3915,E1 17.6804,E2 822.8824} C_DIS
LIN {X 125.1385,Y -26.5004,Z 153,A -12.9763,B 17.5204,C -0.3933,E1 17.6812,E2 821.5492} C_DIS
LIN {X 125.7527,Y -23.4159,Z 153,A -11.5497,B 17.5203,C -0.3983,E1 17.6819,E2 820.1185} C_DIS
LIN {X 126.2886,Y -20.3326,Z 153,A -10.1501,B 17.5202,C -0.4025,E1 17.6826,E2 818.7172} C_DIS
LIN {X 126.7007,Y -17.576,Z 153,A -8.9089,B 17.5201,C -0.4061,E1 17.6831,E2 817.475} C_DIS
LIN {X 127.1328,Y -14.1116,Z 153,A -7.339,B 17.52,C -0.4111,E1 17.6836,E2 815.9022} C_DIS
LIN {X 127.4394,Y -10.9987,Z 153,A -6.0687,B 17.52,C -0.4104,E1 17.6839,E2 814.6452} C_DIS
LIN {X 127.6466,Y -8.2606,Z 153,A -4.6521,B 17.5197,C -0.4213,E1 17.6842,E2 813.2051} C_DIS
LIN {X 127.8109,Y -5.1125,Z 153,A -3.2878,B 17.5197,C -0.4239,E1 17.6844,E2 811.8444} C_DIS
LIN {X 127.9081,Y -1.2237,Z 153,A -1.3727,B 17.5194,C -0.4358,E1 17.6844,E2 809.9067} C_DIS
LIN {X 127.8758,Y 3.1169,Z 153,A 0.3958,B 17.5194,C -0.4351,E1 17.6844,E2 808.1562} C_DIS
LIN {X 127.7076,Y 7.2704,Z 153,A 2.2776,B 17.5193,C -0.4415,E1 17.6841,E2 806.2696} C_DIS
LIN {X 127.4426,Y 10.9613,Z 153,A 3.7323,B 17.5193,C -0.4389,E1 17.6838,E2 804.8364} C_DIS
LIN {X 127.1777,Y 13.6942,Z 153,A 5.0159,B 17.5192,C -0.4447,E1 17.6834,E2 803.5448} C_DIS
LIN {X 126.7615,Y 17.1316,Z 153,A 6.544,B 17.5191,C -0.4485,E1 17.6829,E2 802.0174} C_DIS
LIN {X 126.3305,Y 20.0634,Z 153,A 7.857,B 17.5191,C -0.452,E1 17.6823,E2 800.7045} C_DIS
LIN {X 125.7545,Y 23.4067,Z 153,A 9.3147,B 17.5189,C -0.4542,E1 17.6816,E2 799.252} C_DIS
LIN {X 125.1439,Y 26.4756,Z 153,A 10.6669,B 17.5189,C -0.4565,E1 17.6809,E2 797.9038} C_DIS
LIN {X 124.5461,Y 29.1621,Z 153,A 11.9835,B 17.5187,C -0.4633,E1 17.68,E2 796.576} C_DIS
LIN {X 123.7823,Y 32.2512,Z 153,A 13.3822,B 17.5187,C -0.4665,E1 17.6791,E2 795.1786} C_DIS
LIN {X 122.9551,Y 35.2729,Z 153,A 14.9905,B 17.5183,C -0.4784,E1 17.6778,E2 793.5448} C_DIS
LIN {X 121.5764,Y 39.7651,Z 153,A 16.8405,B 17.5184,C -0.4748,E1 17.6763,E2 791.7221} C_DIS
LIN {X 120.5584,Y 42.7522,Z 153,A 18.28,B 17.5183,C -0.4798,E1 17.675,E2 790.2779} C_DIS
LIN {X 119.4755,Y 45.6915,Z 153,A 19.6709,B 17.5182,C -0.4833,E1 17.6736,E2 788.887} C_DIS
LIN {X 118.1717,Y 48.9612,Z 153,A 21.3852,B 17.5179,C -0.493,E1 17.6718,E2 787.1548} C_DIS
LIN {X 116.4516,Y 52.9266,Z 153,A 23.264,B 17.5179,C -0.4961,E1 17.6697,E2 785.2808} C_DIS
LIN {X 114.9637,Y 56.0826,Z 153,A 24.6988,B 17.5179,C -0.4955,E1 17.6679,E2 783.8592} C_DIS
LIN {X 113.543,Y 58.9066,Z 153,A 26.0533,B 17.5179,C -0.497,E1 17.6662,E2 782.5104} C_DIS
LIN {X 112.0624,Y 61.6783,Z 153,A 27.5042,B 17.5177,C -0.5023,E1 17.6643,E2 781.0532} C_DIS
LIN {X 110.6997,Y 64.0911,Z 153,A 28.8047,B 17.5175,C -0.5078,E1 17.6625,E2 779.7447} C_DIS
LIN {X 109.1375,Y 66.7169,Z 153,A 30.1914,B 17.5175,C -0.512,E1 17.6605,E2 778.3546} C_DIS
LIN {X 106.9186,Y 70.2178,Z 153,A 32.0545,B 17.5173,C -0.5169,E1 17.6576,E2 776.489} C_DIS
LIN {X 104.8133,Y 73.3238,Z 153,A 33.6156,B 17.5173,C -0.5165,E1 17.6552,E2 774.9404} C_DIS
LIN {X 102.9995,Y 75.85,Z 153,A 35.073,B 17.5171,C -0.5223,E1 17.6528,E2 773.4744} C_DIS
LIN {X 100.3583,Y 79.3124,Z 153,A 37.0668,B 17.5169,C -0.5285,E1 17.6493,E2 771.4741} C_DIS
LIN {X 97.7563,Y 82.4981,Z 153,A 38.8936,B 17.5169,C -0.5321,E1 17.6461,E2 769.6478} C_DIS
LIN {X 94.9035,Y 85.7642,Z 153,A 40.8402,B 17.5167,C -0.5365,E1 17.6425,E2 767.6993} C_DIS
LIN {X 92.1066,Y 88.7613,Z 153,A 42.6549,B 17.5166,C -0.5397,E1 17.639,E2 765.8859} C_DIS
LIN {X 89.0049,Y 91.8707,Z 153,A 44.5612,B 17.5166,C -0.5415,E1 17.6352,E2 763.9855} C_DIS
LIN {X 85.8979,Y 94.7821,Z 153,A 46.4828,B 17.5164,C -0.5458,E1 17.6312,E2 762.0612} C_DIS
LIN {X 82.4967,Y 97.7575,Z 153,A 48.4658,B 17.5164,C -0.5481,E1 17.627,E2 760.0818} C_DIS
LIN {X 79.3221,Y 100.3507,Z 153,A 50.254,B 17.5163,C -0.5497,E1 17.6232,E2 758.2983} C_DIS
LIN {X 76.1995,Y 102.7414,Z 153,A 51.9627,B 17.5163,C -0.5509,E1 17.6194,E2 756.5949} C_DIS
LIN {X 73.6589,Y 104.5776,Z 153,A 53.3567,B 17.5162,C -0.5529,E1 17.6162,E2 755.2015} C_DIS
LIN {X 71.0713,Y 106.3531,Z 153,A 54.8219,B 17.5161,C -0.5573,E1 17.6128,E2 753.7289} C_DIS
LIN {X 67.5805,Y 108.6047,Z 153,A 56.6423,B 17.5161,C -0.5587,E1 17.6085,E2 751.9125} C_DIS
LIN {X 64.7473,Y 110.3172,Z 153,A 58.1425,B 17.5159,C -0.5615,E1 17.6049,E2 750.4099} C_DIS
LIN {X 62.0455,Y 111.8591,Z 153,A 59.4652,B 17.5159,C -0.5609,E1 17.6017,E2 749.095} C_DIS
LIN {X 59.3596,Y 113.3051,Z 153,A 60.8567,B 17.5159,C -0.5637,E1 17.5983,E2 747.7003} C_DIS
LIN {X 56.7659,Y 114.6266,Z 153,A 62.2077,B 17.5158,C -0.567,E1 17.5949,E2 746.3436} C_DIS
LIN {X 53.2706,Y 116.293,Z 153,A 63.8632,B 17.5158,C -0.5662,E1 17.5907,E2 744.6969} C_DIS
LIN {X 50.7292,Y 117.423,Z 153,A 65.1586,B 17.5157,C -0.5694,E1 17.5874,E2 743.3958} C_DIS
LIN {X 47.5099,Y 118.7625,Z 153,A 66.6588,B 17.5157,C -0.5688,E1 17.5835,E2 741.9026} C_DIS
LIN {X 44.5974,Y 119.8865,Z 153,A 68.0518,B 17.5157,C -0.57,E1 17.5799,E2 740.5101} C_DIS
LIN {X 41.6667,Y 120.9362,Z 153,A 69.3996,B 17.5157,C -0.5696,E1 17.5763,E2 739.1676} C_DIS
LIN {X 38.6362,Y 121.9384,Z 153,A 70.812,B 17.5157,C -0.5702,E1 17.5726,E2 737.7573} C_DIS
LIN {X 35.6215,Y 122.853,Z 153,A 72.2757,B 17.5156,C -0.5731,E1 17.5687,E2 736.2877} C_DIS
LIN {X 32.6,Y 123.6892,Z 153,A 73.6759,B 17.5156,C -0.5739,E1 17.5649,E2 734.8881} C_DIS
LIN {X 29.6268,Y 124.4349,Z 153,A 75.0525,B 17.5156,C -0.5749,E1 17.5612,E2 733.5113} C_DIS
LIN {X 26.5012,Y 125.1384,Z 153,A 76.4452,B 17.5156,C -0.5742,E1 17.5574,E2 732.1237} C_DIS
LIN {X 23.4288,Y 125.7503,Z 153,A 77.8557,B 17.5156,C -0.5751,E1 17.5535,E2 730.7127} C_DIS
LIN {X 20.8555,Y 126.2013,Z 153,A 79.0695,B 17.5154,C -0.5771,E1 17.5501,E2 729.4941} C_DIS
LIN {X 17.5852,Y 126.6993,Z 153,A 80.521,B 17.5154,C -0.5765,E1 17.5461,E2 728.0465} C_DIS
LIN {X 14.118,Y 127.1321,Z 153,A 82.1055,B 17.5154,C -0.5775,E1 17.5417,E2 726.4604} C_DIS
LIN {X 11.0048,Y 127.4389,Z 153,A 83.3846,B 17.5156,C -0.5735,E1 17.5382,E2 725.1957} C_DIS
LIN {X 8.2706,Y 127.6459,Z 153,A 84.8251,B 17.5153,C -0.581,E1 17.5341,E2 723.7315} C_DIS
LIN {X 5.0859,Y 127.8119,Z 153,A 86.2104,B 17.5153,C -0.5795,E1 17.5303,E2 722.3516} C_DIS
LIN {X 1.9734,Y 127.8979,Z 153,A 87.5762,B 17.5153,C -0.5784,E1 17.5265,E2 720.9898} C_DIS
LIN {X -1.188,Y 127.9084,Z 153,A 89.0393,B 17.5153,C -0.5799,E1 17.5224,E2 719.522} C_DIS
LIN {X -4.6508,Y 127.8289,Z 153,A 90.686,B 17.5153,C -0.5828,E1 17.5178,E2 717.8653} C_DIS
LIN {X -9.3814,Y 127.5685,Z 153,A 92.6358,B 17.5155,C -0.5762,E1 17.5124,E2 715.9363} C_DIS
LIN {X -12.0772,Y 127.3416,Z 153,A 93.8465,B 17.5155,C -0.5757,E1 17.509,E2 714.7265} C_DIS
LIN {X -15.0311,Y 127.0267,Z 153,A 95.1694,B 17.5155,C -0.5748,E1 17.5054,E2 713.4052} C_DIS
LIN {X -18.7356,Y 126.5349,Z 153,A 96.8558,B 17.5155,C -0.5743,E1 17.5007,E2 711.7187} C_DIS
LIN {X -21.5028,Y 126.0933,Z 153,A 98.1074,B 17.5155,C -0.5734,E1 17.4973,E2 710.4683} C_DIS
LIN {X -24.5786,Y 125.5304,Z 153,A 99.6042,B 17.5155,C -0.5757,E1 17.4931,E2 708.9617} C_DIS
LIN {X -27.6366,Y 124.8932,Z 153,A 100.9223,B 17.5156,C -0.5719,E1 17.4896,E2 707.6538} C_DIS
LIN {X -30.7145,Y 124.1727,Z 153,A 102.3416,B 17.5156,C -0.5708,E1 17.4857,E2 706.2353} C_DIS
LIN {X -33.7636,Y 123.3782,Z 153,A 103.766,B 17.5156,C -0.57,E1 17.4819,E2 704.8105} C_DIS
LIN {X -37.126,Y 122.4067,Z 153,A 105.3364,B 17.5157,C -0.5686,E1 17.4777,E2 703.241} C_DIS
LIN {X -39.7644,Y 121.5767,Z 153,A 106.5917,B 17.5157,C -0.5678,E1 17.4743,E2 701.9851} C_DIS
LIN {X -42.7289,Y 120.5668,Z 153,A 107.9507,B 17.5158,C -0.5647,E1 17.4707,E2 700.6323} C_DIS
LIN {X -45.6907,Y 119.4758,Z 153,A 109.4015,B 17.5158,C -0.5643,E1 17.4669,E2 699.1786} C_DIS
LIN {X -48.628,Y 118.3108,Z 153,A 110.9366,B 17.5158,C -0.5664,E1 17.4629,E2 697.6312} C_DIS
LIN {X -51.84,Y 116.9376,Z 153,A 112.2509,B 17.5161,C -0.5561,E1 17.4597,E2 696.3468} C_DIS
LIN {X -54.6902,Y 115.6323,Z 153,A 113.8011,B 17.5161,C -0.5589,E1 17.4557,E2 694.7816} C_DIS
LIN {X -57.5071,Y 114.2579,Z 153,A 115.209,B 17.5161,C -0.557,E1 17.4522,E2 693.3747} C_DIS
LIN {X -59.9657,Y 112.9868,Z 153,A 116.5035,B 17.5161,C -0.5569,E1 17.449,E2 692.0753} C_DIS
LIN {X -63.0323,Y 111.3067,Z 153,A 117.9888,B 17.5162,C -0.5517,E1 17.4454,E2 690.6009} C_DIS
LIN {X -65.1956,Y 110.0534,Z 153,A 119.2956,B 17.5162,C -0.556,E1 17.4422,E2 689.2742} C_DIS
LIN {X -68.3825,Y 108.1015,Z 153,A 120.7386,B 17.5164,C -0.5456,E1 17.4388,E2 687.8592} C_DIS
LIN {X -70.9221,Y 106.4526,Z 153,A 122.3281,B 17.5163,C -0.5507,E1 17.435,E2 686.2448} C_DIS
LIN {X -74.6285,Y 103.8882,Z 153,A 124.1353,B 17.5166,C -0.5401,E1 17.431,E2 684.464} C_DIS
LIN {X -77.1584,Y 102.0229,Z 153,A 125.716,B 17.5165,C -0.5429,E1 17.4274,E2 682.8654} C_DIS
LIN {X -80.5417,Y 99.3742,Z 153,A 127.721,B 17.5165,C -0.5417,E1 17.423,E2 680.8536} C_DIS
LIN {X -83.5484,Y 96.8595,Z 153,A 129.4754,B 17.5166,C -0.538,E1 17.4193,E2 679.1016} C_DIS
LIN {X -86.477,Y 94.2541,Z 153,A 131.2328,B 17.5168,C -0.5342,E1 17.4156,E2 677.3462} C_DIS
LIN {X -89.3346,Y 91.5507,Z 153,A 133.0264,B 17.5168,C -0.5313,E1 17.412,E2 675.5514} C_DIS
LIN {X -92.2243,Y 88.6392,Z 153,A 134.8801,B 17.517,C -0.5276,E1 17.4084,E2 673.6983} C_DIS
LIN {X -94.8963,Y 85.7721,Z 153,A 136.6434,B 17.517,C -0.5238,E1 17.4051,E2 671.9364} C_DIS
LIN {X -97.7602,Y 82.4935,Z 153,A 138.5673,B 17.5172,C -0.5182,E1 17.4016,E2 670.0181} C_DIS
LIN {X -100.3548,Y 79.3167,Z 153,A 140.494,B 17.5172,C -0.5165,E1 17.3982,E2 668.0837} C_DIS
LIN {X -102.9537,Y 75.9123,Z 153,A 142.3809,B 17.5174,C -0.5107,E1 17.3951,E2 666.203} C_DIS
LIN {X -105.4772,Y 72.3648,Z 153,A 144.2293,B 17.5177,C -0.5024,E1 17.3921,E2 664.3688} C_DIS
LIN {X -107.2186,Y 69.7588,Z 153,A 145.5806,B 17.5178,C -0.497,E1 17.3901,E2 663.0255} C_DIS
LIN {X -108.7241,Y 67.3886,Z 153,A 146.9145,B 17.5178,C -0.4961,E1 17.3881,E2 661.6848} C_DIS
LIN {X -110.3354,Y 64.7164,Z 153,A 148.2501,B 17.518,C -0.4903,E1 17.3862,E2 660.3582} C_DIS
LIN {X -111.8821,Y 62.0041,Z 153,A 149.729,B 17.518,C -0.489,E1 17.3842,E2 658.8721} C_DIS
LIN {X -113.5318,Y 58.9278,Z 153,A 151.2896,B 17.5182,C -0.4846,E1 17.3821,E2 657.3141} C_DIS
LIN {X -114.7747,Y 56.4658,Z 153,A 152.5534,B 17.5182,C -0.4821,E1 17.3806,E2 656.0488} C_DIS
LIN {X -116.271,Y 53.318,Z 153,A 154.1376,B 17.5183,C -0.4783,E1 17.3787,E2 654.4643} C_DIS
LIN {X -117.4203,Y 50.7354,Z 153,A 155.4656,B 17.5183,C -0.4767,E1 17.3772,E2 653.131} C_DIS
LIN {X -118.7653,Y 47.503,Z 153,A 156.9892,B 17.5185,C -0.4707,E1 17.3756,E2 651.6148} C_DIS
LIN {X -119.8941,Y 44.5772,Z 153,A 158.4053,B 17.5186,C -0.467,E1 17.3742,E2 650.1995} C_DIS
LIN {X -120.9521,Y 41.6211,Z 153,A 159.8566,B 17.5186,C -0.4642,E1 17.3729,E2 648.7451} C_DIS
LIN {X -122.2595,Y 37.6071,Z 153,A 161.7922,B 17.5188,C -0.46,E1 17.3712,E2 646.8071} C_DIS
LIN {X -123.2803,Y 34.1137,Z 153,A 163.3739,B 17.519,C -0.4536,E1 17.37,E2 645.2333} C_DIS
LIN {X -124.0794,Y 31.0824,Z 153,A 164.7899,B 17.519,C -0.4498,E1 17.369,E2 643.818} C_DIS
LIN {X -124.967,Y 27.295,Z 153,A 166.6498,B 17.519,C -0.4482,E1 17.3679,E2 641.9472} C_DIS
LIN {X -125.7544,Y 23.4073,Z 153,A 168.3189,B 17.5193,C -0.4394,E1 17.367,E2 640.293} C_DIS
LIN {X -126.2909,Y 20.3188,Z 153,A 169.7468,B 17.5193,C -0.4359,E1 17.3663,E2 638.8644} C_DIS
LIN {X -126.7002,Y 17.5791,Z 153,A 171.0022,B 17.5195,C -0.4325,E1 17.3658,E2 637.6091} C_DIS
LIN {X -127.1334,Y 14.1059,Z 153,A 172.6056,B 17.5195,C -0.4288,E1 17.3653,E2 636.0038} C_DIS
LIN {X -127.4405,Y 10.9853,Z 153,A 173.9077,B 17.5197,C -0.4213,E1 17.365,E2 634.7153} C_DIS
LIN {X -127.6502,Y 8.2017,Z 153,A 175.238,B 17.5197,C -0.42,E1 17.3647,E2 633.3777} C_DIS
LIN {X -127.8436,Y 4.2715,Z 153,A 177.2522,B 17.5197,C -0.4224,E1 17.3645,E2 631.3372} C_DIS
LIN {X -127.9142,Y -0.0018,Z 153,A 179.0878,B 17.5199,C -0.4141,E1 17.3645,E2 629.5132} C_DIS
LIN {X -127.8434,Y -4.2782,Z 153,A -178.9421,B 17.52,C -0.4099,E1 17.3645,E2 627.5396} C_DIS
LIN {X -127.6946,Y -7.4802,Z 153,A -177.553,B 17.5201,C -0.4041,E1 17.3648,E2 626.1577} C_DIS
LIN {X -127.4419,Y -10.9696,Z 153,A -176.1157,B 17.5203,C -0.3952,E1 17.3651,E2 624.7373} C_DIS
LIN {X -127.1745,Y -13.7244,Z 153,A -174.8002,B 17.5203,C -0.3938,E1 17.3655,E2 623.4147} C_DIS
LIN {X -126.8315,Y -16.597,Z 153,A -173.4057,B 17.5203,C -0.393,E1 17.366,E2 622.0106} C_DIS
LIN {X -126.291,Y -20.3179,Z 153,A -171.8066,B 17.5205,C -0.3852,E1 17.3667,E2 620.4235} C_DIS
LIN {X -125.5289,Y -24.5866,Z 153,A -169.7495,B 17.5205,C -0.3831,E1 17.3677,E2 618.3556} C_DIS
LIN {X -124.8897,Y -27.6529,Z 153,A -168.4216,B 17.5207,C -0.3765,E1 17.3685,E2 617.0381} C_DIS
LIN {X -124.1699,Y -30.7256,Z 153,A -166.9966,B 17.5208,C -0.3727,E1 17.3694,E2 615.6135} C_DIS
LIN {X -123.3787,Y -33.7618,Z 153,A -165.5686,B 17.5208,C -0.3693,E1 17.3704,E2 614.1846} C_DIS
LIN {X -122.0905,Y -38.1591,Z 153,A -163.4492,B 17.521,C -0.3655,E1 17.3722,E2 612.0599} C_DIS
LIN {X -120.9508,Y -41.6248,Z 153,A -161.9824,B 17.5212,C -0.3555,E1 17.3734,E2 610.6141} C_DIS
LIN {X -120.0207,Y -44.2392,Z 153,A -160.6021,B 17.5212,C -0.3563,E1 17.3748,E2 609.2196} C_DIS
LIN {X -118.9019,Y -47.1642,Z 153,A -159.2146,B 17.5212,C -0.3519,E1 17.3762,E2 607.8353} C_DIS
LIN {X -117.6648,Y -50.1699,Z 153,A -157.6404,B 17.5212,C -0.3516,E1 17.3779,E2 606.2491} C_DIS
LIN {X -116.4511,Y -52.9275,Z 153,A -156.3521,B 17.5213,C -0.346,E1 17.3793,E2 604.9693} C_DIS
LIN {X -114.9583,Y -56.0935,Z 153,A -154.8689,B 17.5215,C -0.3391,E1 17.3811,E2 603.4973} C_DIS
LIN {X -113.5421,Y -58.9083,Z 153,A -153.4141,B 17.5215,C -0.3367,E1 17.383,E2 602.0389} C_DIS
LIN {X -112.3593,Y -61.1351,Z 153,A -152.0973,B 17.5215,C -0.3397,E1 17.3847,E2 600.7017} C_DIS
LIN {X -110.6936,Y -64.1017,Z 153,A -150.6155,B 17.5215,C -0.3344,E1 17.3868,E2 599.2262} C_DIS
LIN {X -108.9012,Y -67.102,Z 153,A -149.097,B 17.5217,C -0.3289,E1 17.389,E2 597.7145} C_DIS
LIN {X -107.4243,Y -69.4419,Z 153,A -147.8579,B 17.5217,C -0.3258,E1 17.3908,E2 596.4766} C_DIS
LIN {X -105.4773,Y -72.3646,Z 153,A -146.1483,B 17.5217,C -0.3264,E1 17.3935,E2 594.7526} C_DIS
LIN {X -102.9595,Y -75.9045,Z 153,A -144.2375,B 17.5218,C -0.3206,E1 17.3967,E2 592.8475} C_DIS
LIN {X -100.362,Y -79.3077,Z 153,A -142.2437,B 17.5218,C -0.3186,E1 17.4001,E2 590.8464} C_DIS
LIN {X -97.994,Y -82.2148,Z 153,A -140.6494,B 17.522,C -0.312,E1 17.4029,E2 589.2631} C_DIS
LIN {X -95.4296,Y -85.1783,Z 153,A -138.8774,B 17.522,C -0.3087,E1 17.4062,E2 587.4905} C_DIS
LIN {X -92.7764,Y -88.0613,Z 153,A -137.1092,B 17.522,C -0.3053,E1 17.4095,E2 585.7219} C_DIS
LIN {X -90.0462,Y -90.8505,Z 153,A -135.34,B 17.5221,C -0.3024,E1 17.413,E2 583.9514} C_DIS
LIN {X -87.1331,Y -93.6479,Z 153,A -133.5505,B 17.5221,C -0.2982,E1 17.4167,E2 582.1652} C_DIS
LIN {X -84.2829,Y -96.2214,Z 153,A -131.6913,B 17.5221,C -0.2995,E1 17.4206,E2 580.2908} C_DIS
LIN {X -81.1775,Y -98.8554,Z 153,A -129.8566,B 17.5222,C -0.2965,E1 17.4245,E2 578.4558} C_DIS
LIN {X -77.9341,Y -101.432,Z 153,A -128.0198,B 17.5222,C -0.2926,E1 17.4285,E2 576.622} C_DIS
LIN {X -74.9359,Y -103.6664,Z 153,A -126.458,B 17.5224,C -0.286,E1 17.432,E2 575.074} C_DIS
LIN {X -72.5255,Y -105.3669,Z 153,A -125.089,B 17.5224,C -0.2855,E1 17.4352,E2 573.6999} C_DIS
LIN {X -70.0182,Y -107.05,Z 153,A -123.6996,B 17.5224,C -0.2846,E1 17.4384,E2 572.3068} C_DIS
LIN {X -67.4262,Y -108.7006,Z 153,A -122.3892,B 17.5224,C -0.2803,E1 17.4415,E2 571.0045} C_DIS
LIN {X -64.4355,Y -110.5003,Z 153,A -120.6628,B 17.5224,C -0.2836,E1 17.4457,E2 569.2595} C_DIS
LIN {X -60.6231,Y -112.6364,Z 153,A -118.7682,B 17.5224,C -0.2789,E1 17.4503,E2 567.3728} C_DIS
LIN {X -57.8392,Y -114.0888,Z 153,A -117.4417,B 17.5226,C -0.2744,E1 17.4536,E2 566.0557} C_DIS
LIN {X -54.684,Y -115.6353,Z 153,A -115.7305,B 17.5226,C -0.2772,E1 17.4579,E2 564.3288} C_DIS
LIN {X -50.7428,Y -117.4171,Z 153,A -113.861,B 17.5226,C -0.2728,E1 17.4627,E2 562.4674} C_DIS
LIN {X -47.5198,Y -118.7585,Z 153,A -112.3514,B 17.5226,C -0.2694,E1 17.4666,E2 560.9642} C_DIS
LIN {X -44.608,Y -119.8825,Z 153,A -110.9856,B 17.5226,C -0.267,E1 17.4701,E2 559.6022} C_DIS
LIN {X -41.6169,Y -120.9535,Z 153,A -109.5813,B 17.5227,C -0.2651,E1 17.4738,E2 558.2001} C_DIS
LIN {X -38.9085,Y -121.8514,Z 153,A -108.2558,B 17.5227,C -0.2657,E1 17.4774,E2 556.869} C_DIS
LIN {X -35.6255,Y -122.8518,Z 153,A -106.7032,B 17.5227,C -0.2652,E1 17.4815,E2 555.3144} C_DIS
LIN {X -32.8241,Y -123.6295,Z 153,A -105.3665,B 17.5227,C -0.2655,E1 17.4851,E2 553.9736} C_DIS
LIN {X -29.564,Y -124.45,Z 153,A -103.8927,B 17.5227,C -0.2636,E1 17.4891,E2 552.5033} C_DIS
LIN {X -26.5071,Y -125.1371,Z 153,A -102.5206,B 17.5227,C -0.2618,E1 17.4929,E2 551.1347} C_DIS
LIN {X -23.6797,Y -125.7023,Z 153,A -101.2056,B 17.5227,C -0.2621,E1 17.4965,E2 549.8166} C_DIS
LIN {X -20.3329,Y -126.2885,Z 153,A -99.6824,B 17.5227,C -0.2616,E1 17.5007,E2 548.293} C_DIS
LIN {X -17.6064,Y -126.6963,Z 153,A -98.442,B 17.5227,C -0.2615,E1 17.5041,E2 547.0515} C_DIS
LIN {X -14.1447,Y -127.1293,Z 153,A -96.8592,B 17.5227,C -0.2619,E1 17.5085,E2 545.4658} C_DIS
LIN {X -10.1237,Y -127.5133,Z 153,A -94.9703,B 17.5227,C -0.2645,E1 17.5138,E2 543.567} C_DIS
LIN {X -6.3766,Y -127.7539,Z 153,A -93.3942,B 17.5227,C -0.2608,E1 17.5181,E2 542.0024} C_DIS
LIN {X -3.1695,Y -127.8743,Z 153,A -91.9876,B 17.5227,C -0.2598,E1 17.5221,E2 540.5989} C_DIS
LIN {X -0.0079,Y -127.915,Z 153,A -90.4986,B 17.5227,C -0.2625,E1 17.5262,E2 539.1007} C_DIS
LIN {X -0.0079,Y -127.915,Z 153,A -90.4986,B 17.5227,C -0.2625,E1 17.5262,E2 539.1007} C_DIS
Enddeposition()
LIN {X 0.9521,Y -134.7809,Z 154,A -92.2463,B 24.9681,C -1.3044,E1 25.0027,E2 538.7959} C_DIS
Startdeposition()
$VEL.CP = VEL_PRINT
LIN {X 5.1254,Y -134.6867,Z 154,A -90.5218,B 24.9682,C -1.3023,E1 25.0075,E2 537.0769} C_DIS
LIN {X 9.0318,Y -134.4832,Z 154,A -88.7613,B 24.9679,C -1.3083,E1 25.0124,E2 535.3029} C_DIS
LIN {X 12.8763,Y -134.1676,Z 154,A -87.2312,B 24.9682,C -1.3032,E1 25.0166,E2 533.7857} C_DIS
LIN {X 16.6858,Y -133.7491,Z 154,A -85.4915,B 24.9678,C -1.3102,E1 25.0215,E2 532.0308} C_DIS
LIN {X 20.3964,Y -133.2319,Z 154,A -84.0434,B 24.9682,C -1.3035,E1 25.0255,E2 530.5998} C_DIS
LIN {X 23.6393,Y -132.6947,Z 154,A -82.6198,B 24.9681,C -1.3061,E1 25.0294,E2 529.1716} C_DIS
LIN {X 27.0355,Y -132.0447,Z 154,A -81.1158,B 24.9679,C -1.3092,E1 25.0335,E2 527.662} C_DIS
LIN {X 31.2213,Y -131.1184,Z 154,A -79.3001,B 24.9679,C -1.3106,E1 25.0385,E2 525.8455} C_DIS
LIN {X 37.2353,Y -129.5401,Z 154,A -76.7744,B 24.968,C -1.307,E1 25.0453,E2 523.3324} C_DIS
LIN {X 42.331,Y -127.9641,Z 154,A -74.4286,B 24.9677,C -1.3141,E1 25.0515,E2 520.9741} C_DIS
LIN {X 46.9537,Y -126.3412,Z 154,A -72.3523,B 24.9675,C -1.3165,E1 25.057,E2 518.8963} C_DIS
LIN {X 49.9668,Y -125.1805,Z 154,A -70.9736,B 24.9675,C -1.3188,E1 25.0606,E2 517.5153} C_DIS
LIN {X 53.3511,Y -123.7752,Z 154,A -69.4862,B 24.9675,C -1.3173,E1 25.0644,E2 516.035} C_DIS
LIN {X 56.3323,Y -122.4473,Z 154,A -68.0355,B 24.9672,C -1.323,E1 25.0681,E2 514.5745} C_DIS
LIN {X 59.2202,Y -121.0776,Z 154,A -66.6961,B 24.9672,C -1.3241,E1 25.0715,E2 513.2359} C_DIS
LIN {X 62.422,Y -119.4578,Z 154,A -65.1714,B 24.967,C -1.3267,E1 25.0752,E2 511.7092} C_DIS
LIN {X 65.8918,Y -117.5816,Z 154,A -63.3142,B 24.9664,C -1.3398,E1 25.0798,E2 509.8266} C_DIS
LIN {X 70.0959,Y -115.1254,Z 154,A -61.3897,B 24.9666,C -1.3356,E1 25.0844,E2 507.9179} C_DIS
LIN {X 73.755,Y -112.8162,Z 154,A -59.546,B 24.9664,C -1.3395,E1 25.0888,E2 506.0711} C_DIS
LIN {X 77.3117,Y -110.4092,Z 154,A -57.639,B 24.966,C -1.3478,E1 25.0932,E2 504.1509} C_DIS
LIN {X 81.1254,Y -107.6374,Z 154,A -55.7282,B 24.966,C -1.3469,E1 25.0974,E2 502.249} C_DIS
LIN {X 84.5894,Y -104.937,Z 154,A -53.8773,B 24.9659,C -1.3502,E1 25.1015,E2 500.3973} C_DIS
LIN {X 87.933,Y -102.1515,Z 154,A -52.0293,B 24.9656,C -1.3544,E1 25.1054,E2 498.5465} C_DIS
LIN {X 91.2935,Y -99.1597,Z 154,A -50.1249,B 24.9654,C -1.3585,E1 25.1094,E2 496.6401} C_DIS
LIN {X 94.5477,Y -96.062,Z 154,A -48.2238,B 24.9652,C -1.3627,E1 25.1132,E2 494.7369} C_DIS
LIN {X 97.667,Y -92.8891,Z 154,A -46.3371,B 24.965,C -1.3673,E1 25.1169,E2 492.8477} C_DIS
LIN {X 100.597,Y -89.7076,Z 154,A -44.4973,B 24.9647,C -1.3721,E1 25.1203,E2 491.0045} C_DIS
LIN {X 103.4297,Y -86.4263,Z 154,A -42.6786,B 24.9645,C -1.3757,E1 25.1236,E2 489.1857} C_DIS
LIN {X 106.181,Y -83.0229,Z 154,A -40.5254,B 24.9634,C -1.3974,E1 25.1274,E2 486.9915} C_DIS
LIN {X 108.4674,Y -80.0127,Z 154,A -39.2164,B 24.9641,C -1.385,E1 25.1295,E2 485.718} C_DIS
LIN {X 110.9562,Y -76.5242,Z 154,A -37.3839,B 24.9638,C -1.3908,E1 25.1325,E2 483.8808} C_DIS
LIN {X 113.5065,Y -72.6871,Z 154,A -35.427,B 24.9635,C -1.3964,E1 25.1355,E2 481.9204} C_DIS
LIN {X 115.957,Y -68.7112,Z 154,A -33.4748,B 24.9633,C -1.4004,E1 25.1383,E2 479.9689} C_DIS
LIN {X 118.1555,Y -64.8579,Z 154,A -31.5906,B 24.963,C -1.406,E1 25.1408,E2 478.0814} C_DIS
LIN {X 119.9621,Y -61.4477,Z 154,A -30.0733,B 24.963,C -1.404,E1 25.1428,E2 476.5766} C_DIS
LIN {X 121.5138,Y -58.3187,Z 154,A -28.6238,B 24.963,C -1.4066,E1 25.1446,E2 475.1288} C_DIS
LIN {X 122.9254,Y -55.2814,Z 154,A -27.1767,B 24.9626,C -1.4123,E1 25.1462,E2 473.6761} C_DIS
LIN {X 124.1859,Y -52.3901,Z 154,A -25.8491,B 24.9625,C -1.4158,E1 25.1477,E2 472.3476} C_DIS
LIN {X 125.5567,Y -49.012,Z 154,A -24.3204,B 24.9623,C -1.4195,E1 25.1493,E2 470.8185} C_DIS
LIN {X 126.7341,Y -45.8819,Z 154,A -22.9038,B 24.962,C -1.4237,E1 25.1506,E2 469.3999} C_DIS
LIN {X 127.8971,Y -42.5322,Z 154,A -21.4278,B 24.9619,C -1.4268,E1 25.152,E2 467.925} C_DIS
LIN {X 129.0149,Y -39.0131,Z 154,A -19.7179,B 24.9612,C -1.4399,E1 25.1534,E2 466.1941} C_DIS
LIN {X 130.1797,Y -34.9279,Z 154,A -18.0897,B 24.9614,C -1.4356,E1 25.1546,E2 464.5852} C_DIS
LIN {X 130.9754,Y -31.8148,Z 154,A -16.6435,B 24.9609,C -1.4447,E1 25.1556,E2 463.126} C_DIS
LIN {X 131.9073,Y -27.7076,Z 154,A -14.8329,B 24.9605,C -1.4517,E1 25.1567,E2 461.3094} C_DIS
LIN {X 132.6294,Y -24.0046,Z 154,A -13.2949,B 24.9605,C -1.4533,E1 25.1574,E2 459.7768} C_DIS
LIN {X 133.2148,Y -20.5071,Z 154,A -11.8351,B 24.9603,C -1.4555,E1 25.1581,E2 458.3202} C_DIS
LIN {X 133.7632,Y -16.5681,Z 154,A -10.1035,B 24.9599,C -1.4635,E1 25.1587,E2 456.5802} C_DIS
LIN {X 134.1622,Y -12.9316,Z 154,A -8.6031,B 24.9598,C -1.4655,E1 25.1592,E2 455.0837} C_DIS
LIN {X 134.4861,Y -8.9849,Z 154,A -6.8279,B 24.9592,C -1.4763,E1 25.1595,E2 453.2936} C_DIS
LIN {X 134.6868,Y -5.1231,Z 154,A -5.2506,B 24.9591,C -1.478,E1 25.1597,E2 451.7217} C_DIS
LIN {X 134.7832,Y -0.718,Z 154,A -3.5476,B 24.9593,C -1.4746,E1 25.1597,E2 450.037} C_DIS
LIN {X 134.7608,Y 2.5222,Z 154,A -1.9664,B 24.9584,C -1.4907,E1 25.1597,E2 448.4272} C_DIS
LIN {X 134.6066,Y 6.9172,Z 154,A -0.1817,B 24.9583,C -1.4921,E1 25.1595,E2 446.6498} C_DIS
LIN {X 134.3308,Y 11.0479,Z 154,A 1.5594,B 24.958,C -1.4968,E1 25.1592,E2 444.9079} C_DIS
LIN {X 133.9663,Y 14.8303,Z 154,A 3.254,B 24.9575,C -1.5066,E1 25.1587,E2 443.2003} C_DIS
LIN {X 133.4861,Y 18.6641,Z 154,A 4.8094,B 24.9575,C -1.507,E1 25.1581,E2 441.6531} C_DIS
LIN {X 132.9485,Y 22.1678,Z 154,A 6.2678,B 24.9573,C -1.5091,E1 25.1574,E2 440.1983} C_DIS
LIN {X 132.2762,Y 25.8853,Z 154,A 7.9825,B 24.9567,C -1.5204,E1 25.1565,E2 438.4669} C_DIS
LIN {X 131.4054,Y 29.9885,Z 154,A 9.6082,B 24.9569,C -1.5172,E1 25.1556,E2 436.8582} C_DIS
LIN {X 130.6546,Y 33.1066,Z 154,A 10.9973,B 24.9565,C -1.523,E1 25.1546,E2 435.4635} C_DIS
LIN {X 129.6101,Y 36.992,Z 154,A 13.0472,B 24.9551,C -1.5476,E1 25.1531,E2 433.3674} C_DIS
LIN {X 128.5676,Y 40.4644,Z 154,A 14.2892,B 24.9558,C -1.5354,E1 25.1521,E2 432.1612} C_DIS
LIN {X 127.2178,Y 44.5246,Z 154,A 16.1369,B 24.9554,C -1.5426,E1 25.1504,E2 430.3069} C_DIS
LIN {X 125.6847,Y 48.6829,Z 154,A 17.83,B 24.9557,C -1.5376,E1 25.1487,E2 428.6351} C_DIS
LIN {X 124.4675,Y 51.7159,Z 154,A 19.2988,B 24.9552,C -1.5462,E1 25.1472,E2 427.1541} C_DIS
LIN {X 123.1844,Y 54.7025,Z 154,A 20.6805,B 24.955,C -1.5503,E1 25.1456,E2 425.7703} C_DIS
LIN {X 121.7122,Y 57.9034,Z 154,A 22.135,B 24.9549,C -1.5522,E1 25.1439,E2 424.3191} C_DIS
LIN {X 120.2262,Y 60.9288,Z 154,A 23.5595,B 24.9546,C -1.5559,E1 25.1421,E2 422.8936} C_DIS
LIN {X 118.5156,Y 64.1977,Z 154,A 25.2341,B 24.954,C -1.5662,E1 25.1399,E2 421.2034} C_DIS
LIN {X 116.4007,Y 67.957,Z 154,A 27.0568,B 24.9538,C -1.5707,E1 25.1374,E2 419.3796} C_DIS
LIN {X 114.0324,Y 71.8592,Z 154,A 28.9512,B 24.9536,C -1.5734,E1 25.1346,E2 417.4885} C_DIS
LIN {X 111.5465,Y 75.6607,Z 154,A 30.8311,B 24.9535,C -1.5756,E1 25.1317,E2 415.6126} C_DIS
LIN {X 109.0162,Y 79.2632,Z 154,A 32.7433,B 24.9531,C -1.5827,E1 25.1286,E2 413.693} C_DIS
LIN {X 106.3222,Y 82.8422,Z 154,A 34.6461,B 24.9528,C -1.5874,E1 25.1253,E2 411.7881} C_DIS
LIN {X 103.5123,Y 86.3279,Z 154,A 36.5725,B 24.9524,C -1.5933,E1 25.1219,E2 409.8566} C_DIS
LIN {X 100.5625,Y 89.7462,Z 154,A 38.4562,B 24.9523,C -1.5959,E1 25.1184,E2 407.9755} C_DIS
LIN {X 97.4491,Y 93.1171,Z 154,A 40.3555,B 24.9522,C -1.5975,E1 25.1148,E2 406.0806} C_DIS
LIN {X 94.3693,Y 96.237,Z 154,A 42.1861,B 24.952,C -1.5997,E1 25.1112,E2 404.2525} C_DIS
LIN {X 91.3724,Y 99.0872,Z 154,A 44.0005,B 24.9516,C -1.6066,E1 25.1075,E2 402.4294} C_DIS
LIN {X 87.9897,Y 102.1026,Z 154,A 45.8736,B 24.9516,C -1.6075,E1 25.1036,E2 400.5613} C_DIS
LIN {X 84.7606,Y 104.7989,Z 154,A 47.6949,B 24.9513,C -1.6128,E1 25.0996,E2 398.7345} C_DIS
LIN {X 81.2091,Y 107.5742,Z 154,A 49.5948,B 24.9511,C -1.6155,E1 25.0954,E2 396.8352} C_DIS
LIN {X 77.4609,Y 110.3042,Z 154,A 51.5528,B 24.9509,C -1.6183,E1 25.091,E2 394.8776} C_DIS
LIN {X 74.0085,Y 112.6494,Z 154,A 53.3163,B 24.9508,C -1.6206,E1 25.0869,E2 393.1144} C_DIS
LIN {X 70.1572,Y 115.088,Z 154,A 55.2886,B 24.9505,C -1.6256,E1 25.0822,E2 391.1366} C_DIS
LIN {X 66.2744,Y 117.3666,Z 154,A 57.1909,B 24.9504,C -1.6278,E1 25.0776,E2 389.2349} C_DIS
LIN {X 62.2222,Y 119.5628,Z 154,A 59.1718,B 24.9501,C -1.6317,E1 25.0727,E2 387.2503} C_DIS
LIN {X 58.3742,Y 121.4872,Z 154,A 60.8649,B 24.9504,C -1.6267,E1 25.0685,E2 385.5736} C_DIS
LIN {X 55.1544,Y 122.9822,Z 154,A 62.3833,B 24.9503,C -1.629,E1 25.0646,E2 384.0535} C_DIS
LIN {X 52.0491,Y 124.3283,Z 154,A 63.7946,B 24.9503,C -1.629,E1 25.061,E2 382.6453} C_DIS
LIN {X 48.9208,Y 125.5922,Z 154,A 65.1918,B 24.9503,C -1.6286,E1 25.0574,E2 381.2525} C_DIS
LIN {X 45.0108,Y 127.0481,Z 154,A 67.2679,B 24.9492,C -1.6465,E1 25.0518,E2 379.1382} C_DIS
LIN {X 40.3254,Y 128.612,Z 154,A 69.1378,B 24.9499,C -1.6359,E1 25.0469,E2 377.297} C_DIS
LIN {X 36.5076,Y 129.7455,Z 154,A 70.7944,B 24.9499,C -1.6352,E1 25.0425,E2 375.6448} C_DIS
LIN {X 33.0839,Y 130.6604,Z 154,A 72.2729,B 24.9499,C -1.6347,E1 25.0385,E2 374.1699} C_DIS
LIN {X 29.7923,Y 131.4502,Z 154,A 73.7452,B 24.9498,C -1.6372,E1 25.0345,E2 372.6935} C_DIS
LIN {X 25.6089,Y 132.329,Z 154,A 75.4845,B 24.95,C -1.6339,E1 25.0298,E2 370.9642} C_DIS
LIN {X 22.4308,Y 132.9046,Z 154,A 76.9682,B 24.9496,C -1.6403,E1 25.0256,E2 369.4668} C_DIS
LIN {X 18.3635,Y 133.529,Z 154,A 78.7828,B 24.9493,C -1.6443,E1 25.0206,E2 367.6446} C_DIS
LIN {X 14.3705,Y 134.0157,Z 154,A 80.3791,B 24.9497,C -1.6386,E1 25.0162,E2 366.0629} C_DIS
LIN {X 10.2136,Y 134.3971,Z 154,A 82.1849,B 24.9496,C -1.6404,E1 25.0112,E2 364.2538} C_DIS
LIN {X 6.5872,Y 134.6231,Z 154,A 83.6909,B 24.9497,C -1.6383,E1 25.007,E2 362.7532} C_DIS
LIN {X 2.5728,Y 134.76,Z 154,A 85.4401,B 24.9496,C -1.6403,E1 25.0021,E2 360.9997} C_DIS
LIN {X -1.5113,Y 134.7776,Z 154,A 87.2287,B 24.9494,C -1.6427,E1 24.9971,E2 359.2055} C_DIS
LIN {X -5.0631,Y 134.6891,Z 154,A 88.6441,B 24.9498,C -1.6373,E1 24.9932,E2 357.8027} C_DIS
LIN {X -9.0289,Y 134.4834,Z 154,A 90.4076,B 24.9496,C -1.6405,E1 24.9882,E2 356.0308} C_DIS
LIN {X -12.7576,Y 134.179,Z 154,A 91.9286,B 24.9498,C -1.6362,E1 24.984,E2 354.5195} C_DIS
LIN {X -16.4642,Y 133.7756,Z 154,A 93.6277,B 24.9495,C -1.6412,E1 24.9793,E2 352.8073} C_DIS
LIN {X -20.4302,Y 133.2267,Z 154,A 95.236,B 24.9499,C -1.6352,E1 24.9749,E2 351.212} C_DIS
LIN {X -24.0308,Y 132.6247,Z 154,A 96.8583,B 24.9497,C -1.6377,E1 24.9704,E2 349.5822} C_DIS
LIN {X -28.2237,Y 131.7959,Z 154,A 98.6066,B 24.9501,C -1.6326,E1 24.9656,E2 347.8439} C_DIS
LIN {X -31.6032,Y 131.0264,Z 154,A 100.0535,B 24.9502,C -1.6298,E1 24.9617,E2 346.4017} C_DIS
LIN {X -34.8027,Y 130.2131,Z 154,A 101.4847,B 24.9502,C -1.6298,E1 24.9578,E2 344.9684} C_DIS
LIN {X -38.5758,Y 129.1476,Z 154,A 103.2533,B 24.95,C -1.6332,E1 24.9531,E2 343.1888} C_DIS
LIN {X -42.3191,Y 127.968,Z 154,A 104.7915,B 24.9506,C -1.6245,E1 24.949,E2 341.6685} C_DIS
LIN {X -45.5548,Y 126.852,Z 154,A 106.2244,B 24.9507,C -1.6215,E1 24.9453,E2 340.2399} C_DIS
LIN {X -48.5228,Y 125.7469,Z 154,A 107.646,B 24.9507,C -1.6235,E1 24.9415,E2 338.8105} C_DIS
LIN {X -51.7722,Y 124.444,Z 154,A 109.114,B 24.9508,C -1.6204,E1 24.9378,E2 337.3468} C_DIS
LIN {X -54.9874,Y 123.0569,Z 154,A 110.5968,B 24.951,C -1.6178,E1 24.934,E2 335.8665} C_DIS
LIN {X -57.8359,Y 121.7444,Z 154,A 111.9218,B 24.9511,C -1.6153,E1 24.9306,E2 334.5442} C_DIS
LIN {X -60.74,Y 120.3223,Z 154,A 113.3503,B 24.9511,C -1.6158,E1 24.927,E2 333.1107} C_DIS
LIN {X -64.0326,Y 118.6046,Z 154,A 115.0163,B 24.951,C -1.6174,E1 24.9229,E2 331.4361} C_DIS
LIN {X -67.8656,Y 116.4541,Z 154,A 116.9074,B 24.9511,C -1.6152,E1 24.9183,E2 329.5447} C_DIS
LIN {X -71.4308,Y 114.3015,Z 154,A 118.6754,B 24.9513,C -1.6117,E1 24.9141,E2 327.7795} C_DIS
LIN {X -75.2453,Y 111.8277,Z 154,A 120.6361,B 24.9515,C -1.6093,E1 24.9096,E2 325.8181} C_DIS
LIN {X -78.3002,Y 109.7097,Z 154,A 122.8248,B 24.9498,C -1.637,E1 24.9045,E2 323.556} C_DIS
LIN {X -82.7777,Y 106.3722,Z 154,A 124.5315,B 24.9522,C -1.5979,E1 24.9009,E2 321.936} C_DIS
LIN {X -86.2138,Y 103.6071,Z 154,A 126.3669,B 24.9525,C -1.5917,E1 24.8969,E2 320.1084} C_DIS
LIN {X -89.9495,Y 100.3804,Z 154,A 128.6216,B 24.9524,C -1.5947,E1 24.8921,E2 317.8377} C_DIS
LIN {X -93.2536,Y 97.3187,Z 154,A 130.4821,B 24.9528,C -1.5873,E1 24.8884,E2 315.9872} C_DIS
LIN {X -96.4405,Y 94.1618,Z 154,A 132.1505,B 24.9538,C -1.5706,E1 24.8851,E2 314.3513} C_DIS
LIN {X -99.4235,Y 91.0065,Z 154,A 134.3109,B 24.9531,C -1.5816,E1 24.881,E2 312.1553} C_DIS
LIN {X -103.5669,Y 86.2623,Z 154,A 136.97,B 24.9536,C -1.5736,E1 24.8761,E2 309.5032} C_DIS
LIN {X -106.7305,Y 82.3155,Z 154,A 139.1172,B 24.954,C -1.5676,E1 24.8724,E2 307.3601} C_DIS
LIN {X -109.2779,Y 78.902,Z 154,A 140.9471,B 24.9542,C -1.5635,E1 24.8694,E2 305.5311} C_DIS
LIN {X -111.7448,Y 75.3677,Z 154,A 142.7511,B 24.9546,C -1.5569,E1 24.8666,E2 303.7339} C_DIS
LIN {X -114.1559,Y 71.6636,Z 154,A 144.692,B 24.9547,C -1.5546,E1 24.8637,E2 301.7889} C_DIS
LIN {X -116.4327,Y 67.9025,Z 154,A 146.5942,B 24.9549,C -1.5507,E1 24.8609,E2 299.8859} C_DIS
LIN {X -118.8036,Y 63.6622,Z 154,A 148.6786,B 24.9552,C -1.5455,E1 24.8582,E2 297.803} C_DIS
LIN {X -120.648,Y 60.0911,Z 154,A 150.3004,B 24.9558,C -1.536,E1 24.8561,E2 296.1951} C_DIS
LIN {X -122.2257,Y 56.8116,Z 154,A 151.8163,B 24.9562,C -1.5297,E1 24.8543,E2 294.6859} C_DIS
LIN {X -123.6365,Y 53.672,Z 154,A 153.0718,B 24.957,C -1.5149,E1 24.8529,E2 293.4588} C_DIS
LIN {X -124.8975,Y 50.6689,Z 154,A 154.712,B 24.9565,C -1.5232,E1 24.8512,E2 291.7898} C_DIS
LIN {X -126.1134,Y 47.5621,Z 154,A 156.044,B 24.957,C -1.5144,E1 24.8498,E2 290.4711} C_DIS
LIN {X -127.2622,Y 44.3965,Z 154,A 158.2224,B 24.9552,C -1.547,E1 24.8478,E2 288.2028} C_DIS
LIN {X -128.8924,Y 39.4133,Z 154,A 159.5142,B 24.9582,C -1.4933,E1 24.8468,E2 287.0315} C_DIS
LIN {X -130.4544,Y 33.8956,Z 154,A 162.2121,B 24.958,C -1.4981,E1 24.8447,E2 284.3064} C_DIS
LIN {X -131.4478,Y 29.8029,Z 154,A 164.117,B 24.958,C -1.498,E1 24.8435,E2 282.3908} C_DIS
LIN {X -132.367,Y 25.4103,Z 154,A 166.0712,B 24.9582,C -1.494,E1 24.8424,E2 280.4345} C_DIS
LIN {X -133.1582,Y 20.8728,Z 154,A 167.961,B 24.9587,C -1.4842,E1 24.8416,E2 278.5569} C_DIS
LIN {X -133.6284,Y 17.6122,Z 154,A 169.3799,B 24.9589,C -1.4805,E1 24.841,E2 277.1384} C_DIS
LIN {X -134.0887,Y 13.6929,Z 154,A 171.1573,B 24.9589,C -1.4798,E1 24.8405,E2 275.3519} C_DIS
LIN {X -134.425,Y 9.8314,Z 154,A 172.7207,B 24.9595,C -1.4702,E1 24.8401,E2 273.802} C_DIS
LIN {X -134.664,Y 5.7062,Z 154,A 174.52,B 24.9597,C -1.4665,E1 24.8399,E2 272.0007} C_DIS
LIN {X -134.767,Y 2.1504,Z 154,A 175.9653,B 24.9602,C -1.4582,E1 24.8398,E2 270.5665} C_DIS
LIN {X -134.7703,Y -1.9519,Z 154,A 177.7694,B 24.9603,C -1.4554,E1 24.8398,E2 268.7581} C_DIS
LIN {X -134.6701,Y -5.5518,Z 154,A 179.4127,B 24.9603,C -1.4559,E1 24.84,E2 267.1038} C_DIS
LIN {X -134.433,Y -9.7218,Z 154,A -178.9269,B 24.9609,C -1.4444,E1 24.8403,E2 265.4608} C_DIS
LIN {X -134.1162,Y -13.4116,Z 154,A -177.2106,B 24.9609,C -1.4463,E1 24.8407,E2 263.7298} C_DIS
LIN {X -133.6527,Y -17.4268,Z 154,A -175.5779,B 24.9613,C -1.4364,E1 24.8413,E2 262.1107} C_DIS
LIN {X -133.0645,Y -21.4724,Z 154,A -173.9065,B 24.9618,C -1.4275,E1 24.842,E2 260.4507} C_DIS
LIN {X -132.2511,Y -26.0154,Z 154,A -171.0594,B 24.9598,C -1.4654,E1 24.8436,E2 257.4963} C_DIS
LIN {X -130.9708,Y -31.8337,Z 154,A -169.2368,B 24.9621,C -1.4218,E1 24.8447,E2 255.7669} C_DIS
LIN {X -129.8814,Y -36.0219,Z 154,A -167.4437,B 24.9626,C -1.4137,E1 24.846,E2 253.9826} C_DIS
LIN {X -128.9639,Y -39.1796,Z 154,A -166.0476,B 24.9628,C -1.4093,E1 24.8471,E2 252.5891} C_DIS
LIN {X -127.9712,Y -42.3097,Z 154,A -164.6309,B 24.963,C -1.406,E1 24.8483,E2 251.172} C_DIS
LIN {X -126.7994,Y -45.7007,Z 154,A -163.1194,B 24.9632,C -1.4007,E1 24.8497,E2 249.6646} C_DIS
LIN {X -125.5284,Y -49.085,Z 154,A -161.5709,B 24.9635,C -1.3967,E1 24.8512,E2 248.1171} C_DIS
LIN {X -123.9852,Y -52.8655,Z 154,A -159.9039,B 24.9639,C -1.3881,E1 24.853,E2 246.4614} C_DIS
LIN {X -121.6199,Y -58.0966,Z 154,A -157.3777,B 24.9641,C -1.3852,E1 24.856,E2 243.9281} C_DIS
LIN {X -120.1411,Y -61.096,Z 154,A -155.9685,B 24.9643,C -1.3805,E1 24.8577,E2 242.5224} C_DIS
LIN {X -118.4714,Y -64.2788,Z 154,A -154.2923,B 24.9641,C -1.3836,E1 24.86,E2 240.83} C_DIS
LIN {X -116.182,Y -68.3292,Z 154,A -152.3857,B 24.9646,C -1.3746,E1 24.8626,E2 238.935} C_DIS
LIN {X -114.0012,Y -71.9088,Z 154,A -150.5465,B 24.9647,C -1.3727,E1 24.8653,E2 237.091} C_DIS
LIN {X -111.4645,Y -75.7818,Z 154,A -148.545,B 24.9649,C -1.3692,E1 24.8684,E2 235.0878} C_DIS
LIN {X -108.8659,Y -79.4702,Z 154,A -146.7782,B 24.9655,C -1.3567,E1 24.8713,E2 233.3422} C_DIS
LIN {X -106.3235,Y -82.8406,Z 154,A -144.8367,B 24.9654,C -1.3596,E1 24.8746,E2 231.3844} C_DIS
LIN {X -103.5488,Y -86.2841,Z 154,A -143.0778,B 24.9659,C -1.3489,E1 24.8777,E2 229.6428} C_DIS
LIN {X -101.3,Y -88.9134,Z 154,A -141.442,B 24.9657,C -1.3538,E1 24.8807,E2 227.9879} C_DIS
LIN {X -98.2471,Y -92.2753,Z 154,A -139.5459,B 24.966,C -1.3477,E1 24.8843,E2 226.0981} C_DIS
LIN {X -94.7389,Y -95.874,Z 154,A -137.3628,B 24.966,C -1.3454,E1 24.8886,E2 223.9111} C_DIS
LIN {X -91.4816,Y -98.9867,Z 154,A -135.4747,B 24.9664,C -1.34,E1 24.8924,E2 222.0282} C_DIS
LIN {X -88.3149,Y -101.8222,Z 154,A -133.6059,B 24.9664,C -1.3395,E1 24.8963,E2 220.1531} C_DIS
LIN {X -84.9318,Y -104.6608,Z 154,A -131.7296,B 24.9666,C -1.3358,E1 24.9004,E2 218.2785} C_DIS
LIN {X -81.4216,Y -107.4139,Z 154,A -129.8164,B 24.9667,C -1.3332,E1 24.9046,E2 216.3645} C_DIS
LIN {X -77.7102,Y -110.1284,Z 154,A -127.8826,B 24.9669,C -1.3287,E1 24.909,E2 214.4347} C_DIS
LIN {X -73.8513,Y -112.7529,Z 154,A -125.8927,B 24.9671,C -1.3258,E1 24.9136,E2 212.4452} C_DIS
LIN {X -70.3137,Y -114.992,Z 154,A -124.1262,B 24.9672,C -1.3223,E1 24.9178,E2 210.6813} C_DIS
LIN {X -66.4897,Y -117.2449,Z 154,A -122.2568,B 24.9674,C -1.3187,E1 24.9223,E2 208.8151} C_DIS
LIN {X -62.977,Y -119.1664,Z 154,A -120.5878,B 24.9676,C -1.3147,E1 24.9264,E2 207.1508} C_DIS
LIN {X -59.807,Y -120.7881,Z 154,A -119.1275,B 24.9679,C -1.3099,E1 24.93,E2 205.6979} C_DIS
LIN {X -56.8531,Y -122.2065,Z 154,A -117.6771,B 24.9678,C -1.3113,E1 24.9337,E2 204.2406} C_DIS
LIN {X -53.7197,Y -123.6159,Z 154,A -116.2264,B 24.9679,C -1.3091,E1 24.9374,E2 202.7916} C_DIS
LIN {X -50.6668,Y -124.8983,Z 154,A -114.8095,B 24.9679,C -1.3081,E1 24.9411,E2 201.3739} C_DIS
LIN {X -48.0342,Y -125.9365,Z 154,A -113.3511,B 24.9673,C -1.3203,E1 24.945,E2 199.8834} C_DIS
LIN {X -43.2187,Y -127.6685,Z 154,A -111.3451,B 24.9679,C -1.3095,E1 24.9502,E2 197.8993} C_DIS
LIN {X -39.7812,Y -128.7798,Z 154,A -109.9095,B 24.9682,C -1.303,E1 24.954,E2 196.4764} C_DIS
LIN {X -36.4288,Y -129.7676,Z 154,A -108.3854,B 24.9682,C -1.304,E1 24.9581,E2 194.9474} C_DIS
LIN {X -33.0485,Y -130.6694,Z 154,A -106.9074,B 24.9682,C -1.3027,E1 24.9621,E2 193.4706} C_DIS
LIN {X -29.2391,Y -131.5765,Z 154,A -105.1506,B 24.968,C -1.3066,E1 24.9669,E2 191.702} C_DIS
LIN {X -25.4994,Y -132.35,Z 154,A -103.6318,B 24.9683,C -1.3004,E1 24.971,E2 190.1962} C_DIS
LIN {X -22.1526,Y -132.951,Z 154,A -102.1512,B 24.9683,C -1.3018,E1 24.9751,E2 188.7108} C_DIS
LIN {X -17.9411,Y -133.5852,Z 154,A -100.3295,B 24.9683,C -1.302,E1 24.9801,E2 186.8873} C_DIS
LIN {X -14.684,Y -133.982,Z 154,A -98.9408,B 24.9683,C -1.3015,E1 24.984,E2 185.499} C_DIS
LIN {X -10.8006,Y -134.3517,Z 154,A -97.2037,B 24.9681,C -1.3056,E1 24.9888,E2 183.7512} C_DIS
LIN {X -6.7356,Y -134.6157,Z 154,A -95.5732,B 24.9683,C -1.3002,E1 24.9934,E2 182.133} C_DIS
LIN {X -2.7095,Y -134.7577,Z 154,A -93.833,B 24.9683,C -1.3019,E1 24.9982,E2 180.3885} C_DIS
LIN {X 0.9521,Y -134.7809,Z 154,A -92.2453,B 24.9682,C -1.304,E1 25.0027,E2 178.7959} C_DIS
Enddeposition()
LIN {X 0.9521,Y -134.7809,Z 154,A -92.2453,B 24.9682,C -1.304,E1 25.0027,E2 178.7959} C_DIS
Startdeposition()
$VEL.CP = VEL_PRINT
LIN {X -0.4991,Y -133.8458,Z 154,A -93.389,B 24.2112,C -1.1345,E1 24.2348,E2 180.2494} C_DIS
LIN {X -4.0061,Y -133.7868,Z 154,A -94.9628,B 24.2114,C -1.1306,E1 24.2303,E2 181.8329} C_DIS
LIN {X -8.2384,Y -133.5926,Z 154,A -96.6754,B 24.2111,C -1.1357,E1 24.2256,E2 183.5337} C_DIS
LIN {X -12.4082,Y -133.2705,Z 154,A -98.4936,B 24.2112,C -1.1343,E1 24.2205,E2 185.3561} C_DIS
LIN {X -16.0057,Y -132.8859,Z 154,A -100.0219,B 24.2112,C -1.1356,E1 24.2163,E2 186.8822} C_DIS
LIN {X -20.1372,Y -132.3232,Z 154,A -101.8254,B 24.2112,C -1.1351,E1 24.2113,E2 188.6884} C_DIS
LIN {X -23.6191,Y -131.7458,Z 154,A -103.2984,B 24.2111,C -1.1375,E1 24.2073,E2 190.1571} C_DIS
LIN {X -27.0283,Y -131.0893,Z 154,A -104.8663,B 24.2112,C -1.134,E1 24.2029,E2 191.7353} C_DIS
LIN {X -31.1791,Y -130.1641,Z 154,A -106.641,B 24.2111,C -1.1373,E1 24.1981,E2 193.5045} C_DIS
LIN {X -34.6412,Y -129.2857,Z 154,A -108.1226,B 24.2109,C -1.1406,E1 24.1941,E2 194.9803} C_DIS
LIN {X -37.69,Y -128.4299,Z 154,A -109.523,B 24.2109,C -1.1393,E1 24.1904,E2 196.3862} C_DIS
LIN {X -41.6611,Y -127.1989,Z 154,A -111.2085,B 24.2107,C -1.1453,E1 24.1859,E2 198.06} C_DIS
LIN {X -47.0449,Y -125.3058,Z 154,A -113.7139,B 24.2107,C -1.1444,E1 24.1793,E2 200.5728} C_DIS
LIN {X -50.2361,Y -124.061,Z 154,A -115.1962,B 24.2107,C -1.1451,E1 24.1754,E2 202.0568} C_DIS
LIN {X -53.4702,Y -122.7022,Z 154,A -116.6785,B 24.2107,C -1.1477,E1 24.1716,E2 203.5364} C_DIS
LIN {X -56.2148,Y -121.4686,Z 154,A -118.0072,B 24.2107,C -1.1472,E1 24.1683,E2 204.8696} C_DIS
LIN {X -59.3011,Y -119.9921,Z 154,A -119.4303,B 24.2105,C -1.151,E1 24.1647,E2 206.2872} C_DIS
LIN {X -62.1115,Y -118.5617,Z 154,A -120.8045,B 24.2105,C -1.1516,E1 24.1613,E2 207.6638} C_DIS
Enddeposition()
END
